(* PLC project HomeAutomation.project, CODESYS CODESYS V3.5 SP21 Patch 3 *)
(* stored: creationDateTime 2026-09-14T20:36:57.2716108, modificationDateTime 2026-09-14T20:35:48.0989634 *)

{attribute 'to_string'}
TYPE E_DIMMER : (idle, soft_turn_on_restore, soft_turn_off, quick_turn_on, quick_turn_off, ramp_up_or_down, low_or_high_entering, low_or_high_leaving, low_or_high_released_by_user, blink);
END_TYPE

TYPE E_DIMMER_CURVE : (linear, logarithmic, cubic);
END_TYPE

(* values of E_RELAY_TYPE: NO: Normally open, and the default. The load is live when the output is TRUE, so a dead PLC leaves it off. What almost every lighting circuit is. Which way round the contact sits decides nothing in the PLC - the output behaves identically either way - and everything in the Home Assistant discovery config, where it swaps the payload_on / payload_off pair so the entity reports the state of the LOAD rather than the state of the coil.; NC: Normally closed. The load is live when the output is FALSE, so a dead PLC leaves it ON - which is the point: sockets, and anything that must survive the controller, are wired this way. Home Assistant reads such an output exactly backwards unless it is told, and no build can catch that, because nothing in the PLC is wrong. *)

{attribute 'qualified_only'}
{attribute 'strict'}
TYPE E_RELAY_TYPE : (NO := 0, NC := 1);
END_TYPE

(* values of E_RS485_DUCO_NODE_TYPE: Unknown: A module type this enumeration does not name, and the value a node holds before the bus has answered for the first time. Zero is deliberately not a Duco type. The manual assigns parameters 01..09 to node 0 and reserves them, so no real component ever reports 0, which leaves it free to mean "not established yet". A node in this state publishes its registers and announces nothing: inventing entities for a component whose layout is unknown would put numbers under labels that were guessed.; DucoBoxFocus: The ventilation unit itself, always node 1. Its register block is the one that is model-specific: read parameters 3, 4 and 5 are current, average and maximum power in watts. A DucoBox Energy or Silent Connect answers those same addresses with something else, which is why this block is named for the Focus.; ValveSensorless: Control valve with no sensor of its own. Reports status, ventilation position and indoor temperature; no CO2 and no humidity.; ValveCO2: Control valve with a CO2 sensor. Adds read parameter 4, the measured CO2 in ppm, and write parameter 1, the CO2 setpoint.; ValveHumidity: Control valve with a humidity sensor. Adds read parameter 5, the relative humidity as a percentage times 100, and write parameters 2 and 3, the RH setpoint and whether delta control is enabled.; UserControl: Wall control, with or without a battery. A battery unit reports no indoor temperature. Its write side collides with the valves': parameters 5 and 6 are the values of buttons 2 and 3 here, where a valve has auto minimum and auto maximum. Anything mapping a holding register to an entity has to branch on the type first.; SensorCO2: CO2 sensor, either a room sensor or a box sensor. A box sensor reports no status and no ventilation position, so its entity set is smaller than a room sensor's even though both answer type 15.; SensorHumidity: Humidity sensor, either a room sensor or a box sensor. Same split as SensorCO2: a box sensor has neither status nor ventilation position.; WindowVentilator: Electronically controlled window ventilator. Two of its registers mean something different from every valve: parameter 2 is the ventilator opening rather than an extraction level, 0 shut to 100 open, and parameter 3 is the OUTDOOR temperature. A reader that assumes "3 is the room temperature" reports the weather as a room.; SwitchSensor: Switch sensor: presence detection, a heat-pump demand input, or an overrule input, selected by write parameter 1. Reports status and ventilation position only.; ActuatorBoard: Actuator board driving a 2/3-point or PWM output. Shares the window ventilator's outdoor temperature on parameter 3, and is the one component where parameter 4 is not CO2 at all: it is the PWM-in percentage. Publishing it as air quality is the mistake this enumeration exists to prevent.; ValveHumidityCO2: Control valve carrying both sensors, and the only type that fills every read parameter: status, position, temperature, CO2 and humidity. Out of sequence at 24 because Duco added it after the 11..19 block was allocated. *)

{attribute 'qualified_only'}
TYPE E_RS485_DUCO_NODE_TYPE : (Unknown := 0, DucoBoxFocus := 10, ValveSensorless := 11, ValveCO2 := 12, ValveHumidity := 13, UserControl := 14, SensorCO2 := 15, SensorHumidity := 16, WindowVentilator := 17, SwitchSensor := 18, ActuatorBoard := 19, ValveHumidityCO2 := 24);
END_TYPE

{attribute 'qualified_only'}
{attribute 'strict'}
{attribute 'to_string'}
TYPE E_HVAC_MODE : (off := 0, auto := 1, heat := 2);
END_TYPE

(* values of E_MQTT_ENTITY: Default: announce as whatever this function block announces by default; Fan: Home Assistant fan platform. Supported by the binary and bistable outputs as an on/off fan; speed and oscillation need topics a binary output has nothing to report on, so they are left out of the published config. *)

{attribute 'qualified_only'}
{attribute 'strict'}
TYPE E_MQTT_ENTITY : (Default := 0, BinarySensor := 1, Sensor := 2, Switch := 3, Light := 4, LightDimmer := 5, Lock := 6, Siren := 7, Valve := 8, Cover := 9, Climate := 10, Event := 11, Fan := 12);
END_TYPE

TYPE MQTT_DISCOVERY_AVTY_T : STRUCT
  topic : JSONVAR;
END_STRUCT;
END_TYPE

TYPE MQTT_DISCOVERY_BASE : STRUCT
  name : JSONVAR;
  default_entity_id : JSONVAR;  (* default entity id *)
  uniq_id : JSONVAR;  (* unique_id *)
  avty : ARRAY[1..2] OF MQTT_DISCOVERY_AVTY_T;  (* availability *)
  avty_mode : JSONVAR;  (* availability mode *)
  pl_avail : JSONVAR;  (* payload_available *)
  pl_not_avail : JSONVAR;  (* payload_not_available *)
  dev : MQTT_DISCOVERY_DEVICE;  (* device *)
  qos : JSONVAR;  (* mqtt qos *)
END_STRUCT;
END_TYPE

TYPE MQTT_DISCOVERY_BINARY_SENSOR : STRUCT
  stat_t : JSONVAR;  (* state_topic *)
  pl_on : JSONVAR;  (* payload_on *)
  pl_off : JSONVAR;  (* payload_off *)
  dev_cla : JSONVAR;  (* device class *)
END_STRUCT;
END_TYPE

TYPE MQTT_DISCOVERY_BINARY_SENSOR_ENT_CAT : STRUCT
  ent_cat : JSONVAR;  (* entity category *)
END_STRUCT;
END_TYPE

TYPE MQTT_DISCOVERY_CLIMATE : STRUCT
  init : JSONVAR;  (* initial desired temperature *)
  curr_temp_t : JSONVAR;  (* current temperature topic *)
  curr_hum_t : JSONVAR;  (* current humidity topic *)
  modes : ARRAY[1..3] OF JSONVAR;  (* modes *)
  mode_cmd_t : JSONVAR;  (* mode command topic *)
  mode_stat_t : JSONVAR;  (* mode state topic *)
  temp_cmd_t : JSONVAR;  (* temperature command topic *)
  temp_stat_t : JSONVAR;  (* temperature state topic *)
  temp_step : JSONVAR;  (* temperature step *)
  opt : JSONVAR;  (* optimistic *)
END_STRUCT;
END_TYPE

TYPE MQTT_DISCOVERY_COVER : STRUCT
  cmd_t : JSONVAR;  (* command_topic *)
  pl_open : JSONVAR;  (* payload open *)
  pl_cls : JSONVAR;  (* payload_close *)
  pl_stop : JSONVAR;  (* payload_stop *)
  stat_t : JSONVAR;  (* state topic *)
  stat_open : JSONVAR;  (* state open *)
  stat_opening : JSONVAR;  (* state opening *)
  stat_clsd : JSONVAR;  (* state closed *)
  stat_closing : JSONVAR;  (* state closing *)
  stat_stopped : JSONVAR;  (* state stopped *)
  opt : JSONVAR;  (* optimistic *)
  dev_cla : JSONVAR;  (* device class *)
END_STRUCT;
END_TYPE

TYPE MQTT_DISCOVERY_COVER_POSITION : STRUCT
  pos_t : JSONVAR;  (* position_topic - where the cover reports how far open it is, as a number between pos_clsd and pos_open. *)
  set_pos_t : JSONVAR;  (* set_position_topic - where Home Assistant asks for a position. Its presence is what puts a slider on the entity rather than three buttons. *)
  pos_open : JSONVAR;  (* position_open - the number that means fully open, normally 100 *)
  pos_clsd : JSONVAR;  (* position_closed - the number that means fully closed, normally 0 *)
END_STRUCT;
END_TYPE

TYPE MQTT_DISCOVERY_DEVICE : STRUCT
  name : JSONVAR;
  cu : JSONVAR;  (* configuration_url *)
  ids : JSONVAR;  (* identifiers *)
  mf : JSONVAR;  (* manufacturer *)
  mdl : JSONVAR;  (* model *)
  sw : JSONVAR;  (* sw_version *)
  hw : JSONVAR;  (* hw_version *)
END_STRUCT;
END_TYPE

TYPE MQTT_DISCOVERY_EVENT : STRUCT
  stat_t : JSONVAR;  (* state topic *)
  evt_typ : ARRAY[1..3] OF JSONVAR;  (* event types *)
  dev_cla : JSONVAR;  (* device class *)
END_STRUCT;
END_TYPE

TYPE MQTT_DISCOVERY_FAN : STRUCT
  cmd_t : JSONVAR;  (* command_topic (REQUIRED) *)
  stat_t : JSONVAR;  (* state_topic *)
  pl_on : JSONVAR;  (* payload_on *)
  pl_off : JSONVAR;  (* payload_off *)
  pct_cmd_t : JSONVAR;  (* percentage_command_topic *)
  pct_stat_t : JSONVAR;  (* percentage_state_topic *)
  spd_rng_min : JSONVAR;  (* speed_range_min *)
  spd_rng_max : JSONVAR;  (* speed_range_max *)
  osc_cmd_t : JSONVAR;  (* oscillation_command_topic *)
  osc_stat_t : JSONVAR;  (* oscillation_state_topic *)
  pl_osc_on : JSONVAR;  (* payload_oscillation_on *)
  pl_osc_off : JSONVAR;  (* payload_oscillation_off *)
  opt : JSONVAR;  (* optimistic *)
END_STRUCT;
END_TYPE

TYPE MQTT_DISCOVERY_LIGHT : STRUCT
  cmd_t : JSONVAR;  (* command_topic *)
  pl_on : JSONVAR;  (* payload_on *)
  pl_off : JSONVAR;  (* payload_off *)
  stat_t : JSONVAR;  (* state_topic *)
  opt : JSONVAR;  (* optimistic *)
END_STRUCT;
END_TYPE

TYPE MQTT_DISCOVERY_LIGHT_DIMMER : STRUCT
  bri_stat_t : JSONVAR;  (* brightness state topic *)
  bri_cmd_t : JSONVAR;  (* brightness command topic *)
  bri_scl : JSONVAR;  (* brightness scale *)
  on_cmd_type : JSONVAR;  (* on command type *)
  dmxChannel : JSONVAR;  (* DMX *)
  dmxWidth : JSONVAR;
  dmxUniverse : JSONVAR;
END_STRUCT;
END_TYPE

TYPE MQTT_DISCOVERY_LOCK : STRUCT
  cmd_t : JSONVAR;  (* command_topic *)
  pl_lock : JSONVAR;  (* payload lock *)
  pl_unlk : JSONVAR;  (* payload unlock *)
  stat_t : JSONVAR;  (* state_topic *)
  stat_locked : JSONVAR;  (* state locked *)
  stat_unlocked : JSONVAR;  (* state unlocked *)
  opt : JSONVAR;  (* optimistic *)
END_STRUCT;
END_TYPE

TYPE MQTT_DISCOVERY_SENSOR : STRUCT
  stat_t : JSONVAR;  (* state_topic *)
  exp_aft : JSONVAR;  (* expire after *)
  dev_cla : JSONVAR;  (* device class, can be null *)
  unit_of_meas : JSONVAR;  (* unit of measurement, can be null *)
  stat_cla : JSONVAR;  (* state class, can be null *)
END_STRUCT;
END_TYPE

TYPE MQTT_DISCOVERY_SENSOR_DIAGNOSTIC : STRUCT
  stat_t : JSONVAR;  (* state_topic *)
  exp_aft : JSONVAR;  (* expire after *)
  ent_cat : JSONVAR;  (* entity category *)
  unit_of_meas : JSONVAR;  (* Added so a diagnostic entity can still carry a unit and keep long-term statistics. A diagnostic sensor is still a sensor: link quality belongs under diagnostics rather than on a dashboard, but it is only worth having if Home Assistant will graph it. Empty on every entity that does not set them, where they serialise as null - the same way stat_cla was added to the ordinary sensor struct. *)
  stat_cla : JSONVAR;
END_STRUCT;
END_TYPE

TYPE MQTT_DISCOVERY_SIREN : STRUCT
  cmd_t : JSONVAR;  (* command_topic *)
  pl_on : JSONVAR;  (* payload_on *)
  pl_off : JSONVAR;  (* payload_off *)
  stat_t : JSONVAR;  (* state_topic *)
  stat_on : JSONVAR;  (* state on *)
  stat_off : JSONVAR;  (* state off *)
  opt : JSONVAR;  (* optimistic *)
END_STRUCT;
END_TYPE

TYPE MQTT_DISCOVERY_SWITCH : STRUCT
  cmd_t : JSONVAR;  (* command_topic *)
  pl_on : JSONVAR;  (* payload_on *)
  pl_off : JSONVAR;  (* payload_off *)
  stat_t : JSONVAR;  (* state_topic *)
  stat_on : JSONVAR;  (* state on *)
  stat_off : JSONVAR;  (* state off *)
  opt : JSONVAR;  (* optimistic *)
  dev_cla : JSONVAR;  (* device class *)
END_STRUCT;
END_TYPE

TYPE MQTT_DISCOVERY_VALVE : STRUCT
  cmd_t : JSONVAR;  (* command topic *)
  pl_open : JSONVAR;  (* payload open *)
  pl_cls : JSONVAR;  (* payload_close *)
END_STRUCT;
END_TYPE

TYPE MQTT_DISCOVERY_VALVE_STATE : STRUCT
  stat_t : JSONVAR;  (* state_topic *)
  stat_clsd : JSONVAR;  (* state clsoed *)
  stat_open : JSONVAR;  (* state closing stat_closing: JSONVAR; state open *)
  opt : JSONVAR;  (* state opening stat_opening: JSONVAR; optimistic *)
  dev_cla : JSONVAR;  (* device class *)
END_STRUCT;
END_TYPE

TYPE ST_MQTT_MESSAGE : STRUCT
  Payload : STRING(1500);
  Topic : STRING(GVL_MQTT.MQTT_TOPIC_LEN);
  Qos : MQTT.QoS;
  MqttRetain : BOOL;
END_STRUCT;
END_TYPE

TYPE MQTT_DISCOVERY_BUTTON : STRUCT
  cmd_t : JSONVAR;  (* command_topic *)
  pl_prs : JSONVAR;  (* payload_press - what is sent when the button is pressed *)
  ent_cat : JSONVAR;  (* entity_category, can be null *)
  dev_cla : JSONVAR;  (* device_class - only identify, restart and update exist for a button; usually null *)
END_STRUCT;
END_TYPE

TYPE MQTT_DISCOVERY_NUMBER : STRUCT
  cmd_t : JSONVAR;  (* command_topic *)
  stat_t : JSONVAR;  (* state_topic - the value the device actually holds, read back rather than assumed *)
  min_val : JSONVAR;  (* min - signed, because a release-the-override value of -1 is a real setting *)
  max_val : JSONVAR;  (* max *)
  step : JSONVAR;  (* step *)
  unit_of_meas : JSONVAR;  (* unit_of_measurement, can be null *)
  mode : JSONVAR;  (* mode - 'box' or 'slider'. A slider on a 0-2000 ppm setpoint is unusable, so this is per entity *)
  dev_cla : JSONVAR;  (* device_class, can be null *)
  ent_cat : JSONVAR;  (* entity_category - 'config' keeps a setpoint out of the main dashboard *)
  opt : JSONVAR;  (* optimistic - FALSE wherever a state topic exists *)
END_STRUCT;
END_TYPE

TYPE A_RS485_READ_BUFFER : ARRAY[0..124] OF WORD;
END_TYPE

TYPE A_RS485_STEP_LIST : ARRAY[0..7] OF ST_RS485_STEP;
END_TYPE

TYPE E_RS485_EASTRON_SDM_DEVICE : (SDM120, SDM220, SDM630);
END_TYPE

(* values of E_RS485_STEP_STATE: IDLE: No step in flight. Start() will be accepted.; BUSY: Transmitting, or waiting for the line to go quiet.; OK: A reply arrived, addressed to us, with the function code we asked for and a CRC of zero over the whole trimmed frame. For a read, ReadBuffer holds Registers() words. Reported for one cycle, then the transport returns to IDLE.; FAILED: No reply, a bad CRC, the wrong slave, the wrong function code, or a Modbus exception reply. Which of those it was is in the transport's counters, not in this value - the scheduler does not need to care and the counters are how a line fault is diagnosed without a scope. *)

{attribute 'qualified_only'}
{attribute 'strict'}
TYPE E_RS485_STEP_STATE : (IDLE := 0, BUSY := 1, OK := 2, FAILED := 3);
END_TYPE

(* values of E_RS485_WORK_LEVEL: NONE: Nothing to do. The scheduler passes over this device.; POLL: A routine read whose interval timer has elapsed. Served round-robin, after every pending COMMAND.; COMMAND: Something a person or Home Assistant asked for, so latency is visible. Served before any POLL, but still round-robin among themselves, so a chatty device cannot starve a quiet one. *)

{attribute 'qualified_only'}
{attribute 'strict'}
TYPE E_RS485_WORK_LEVEL : (NONE := 0, POLL := 1, COMMAND := 2);
END_TYPE

TYPE ST_RS485_COMMISSION_REQUEST : STRUCT
  DeviceId : BYTE;  (* Address the device answers on. Its own, not a guess: a device that has to be hunted for is found by rate and framing, never by walking addresses. *)
  ProbeFunction : BYTE;  (* Function code for the probe read. 3 for holding registers, 4 for input. *)
  ProbeAddress : UINT;  (* Register to read as the probe. Any register that always answers will do - the reply is never decoded, it only has to arrive. *)
  ProbeQuantity : UINT;  (* How many registers the probe asks for. *)
  WriteFunction : BYTE;  (* Function code for the correction. 6 for a single holding register. *)
  WriteAddress : UINT;  (* Register holding the setting that has to change - the device's baud rate, in the only case that exists so far. *)
  WriteValue : WORD;  (* Value that puts the device on this bus. The device encodes it, because only the device knows whether its register takes a rate, a code or an index. *)
  Bauds : ARRAY[0..15] OF UDINT;  (* Rates to try, in the order worth trying them, and how many of them are filled. Put the bus rate first: a device that is already commissioned then costs one Modbus exchange and the sweep ends there. *)
  BaudCount : INT;
  StopBits : ARRAY[0..3] OF BYTE;  (* Framing codes to try, same idea. 255 means leave the port's own framing, which is the ordinary case; 1..3 force the raw SysCom code, because the enumerator names are not portable across runtimes. *)
  StopCount : INT;
  ReportTopic : STRING(32);  (* Topic suffix for the retained result, under the bus prefix. Empty publishes nothing. *)
END_STRUCT;
END_TYPE

TYPE ST_RS485_STEP : STRUCT
  DeviceId : BYTE;  (* Modbus unit id of the slave this step addresses. *)
  FunctionCode : BYTE;  (* 3 read holding, 4 read input, 6 write single, 16 write multiple. Anything else is rejected by the transport rather than guessed at. *)
  Address : UINT;  (* First register, read or write. One field, because a step is only ever one or the other. *)
  Quantity : UINT;  (* Registers to read, or to write. Ignored by FC6, which is always one. *)
  Data : ARRAY[0..7] OF WORD;  (* Payload for a write step. Eight registers is the most an FC16 frame may carry here, which bounds the transmit buffer at 9 + 2*8 = 25 bytes. *)
  AbortOnError : BOOL;  (* TRUE skips the remaining steps of the transaction if this one fails. Set it on the write of a read-after-write: publishing a read-back that never happened, after a write that failed, is the exact inaccuracy the pairing exists to remove. FALSE - the default - suits a batch of independent reads, where one failing register block should not cost the others. *)
END_STRUCT;
END_TYPE

INTERFACE I_RS485_DEVICE
METHOD OnTransactionDone
  VAR_INPUT
    StepsRun : INT;  (* Steps actually executed. Fewer than requested means an AbortOnError step failed. *)
    Failures : INT;  (* How many of those failed. Zero is the only wholly good outcome. *)
  END_VAR
END_METHOD
METHOD OnStepResult
  VAR_INPUT
    StepIndex : INT;  (* Which step of the transaction this is the answer to, indexed as BuildTransaction filled it. Passed in rather than remembered, which is what retires the ActiveRtuQuery and ActiveNode tags every device block used to keep. *)
    Failed : BOOL;  (* No reply, a bad frame, or a Modbus exception. pData holds nothing meaningful. *)
    pData : POINTER TO A_RS485_READ_BUFFER;  (* Registers returned by a read step, big-endian, index 0 being the first register requested. Meaningless for a write step and after a failure. *)
    Count : INT;  (* How many registers pData actually holds. A device that trusts this rather than the quantity it asked for cannot read past the end of a short reply. *)
  END_VAR
END_METHOD
METHOD BuildTransaction : INT
  VAR_INPUT
    pSteps : POINTER TO A_RS485_STEP_LIST;  (* Scheduler-owned scratch. Fill entries 0..n-1 and return n; the memory is only valid for the duration of this call. *)
  END_VAR
END_METHOD
METHOD HasWork : E_RS485_WORK_LEVEL
END_METHOD
METHOD GetCommissioning : BOOL
  VAR_INPUT
    BusBaudrate : UDINT;
    pRequest : POINTER TO ST_RS485_COMMISSION_REQUEST;
  END_VAR
END_METHOD
END_INTERFACE

INTERFACE I_RS485_TRANSPORT
METHOD Registers : INT
END_METHOD
METHOD ReadBuffer : POINTER TO A_RS485_READ_BUFFER
END_METHOD
METHOD Service : E_RS485_STEP_STATE
END_METHOD
METHOD Start : BOOL
  VAR_INPUT
    pStep : POINTER TO ST_RS485_STEP;
  END_VAR
END_METHOD
METHOD Retune : BOOL
  VAR_INPUT
    Baudrate : UDINT;  (* 0 keeps the configured rate *)
    StopBitsRaw : BYTE;  (* 255 keeps the configured framing *)
    ReplyTimeout : TIME;  (* T#0S keeps the configured timeout *)
    GapTime : TIME;  (* T#0S keeps the configured gap *)
  END_VAR
END_METHOD
METHOD RestoreTuning
END_METHOD
METHOD LastRxCount : UDINT
END_METHOD
END_INTERFACE

{attribute 'reflection'}
FUNCTION_BLOCK FB_INPUT_BINARYSENSOR_MQTT EXTENDS FB_MQTT_BASE
  VAR_OUTPUT
    Q : BOOL;  (* Follows the input but debounced *)
    EVENT : BOOL;  (* Event outputs only high for on clock cycle *)
    EVENT_R : BOOL;
    EVENT_F : BOOL;
  END_VAR
  VAR
    {attribute 'noinit'}
    {attribute 'instance-path'}
    sInstancePath : STRING(GVL_MQTT.MQTT_TOPIC_LEN);  (* object's full instance name *)
    bStartup : BOOL := TRUE;
    fbDebounce : OSCAT_BUILDING.DEBOUNCE;  (* to debounce the physical input *)
    fbRTrig : Standard.R_TRIG;  (* to detect a rising edge on the debounced signal *)
    fbFTrig : Standard.F_TRIG;  (* to detect a falling edge on the debounced signal *)
    T_TurnOffDelay : TIME := TIME#0ms;
    fbTurnOffDelayTimer : OSCAT_BASIC.TOF;
  END_VAR
  VAR_INPUT
    BS : BOOL;
    ProcessImageValid : BOOL := TRUE;  (* TRUE once the K-bus has finished starting and the mapped inputs mean something. FALSE holds this sensor at rest. Defaulted TRUE so no existing call site changes behaviour, but pass Pfc200Bus.xConfigFinished on anything whose loop is normally CLOSED. Until the bus is up every mapped word reads zero, and on an inverted loop zero IS the alarm - so a fire sensor left ungated raises its alarm on every single cold start, deterministically. That is not a plausible-looking value like an RTD's 0.0 C; it is the tripped state itself. *)
  END_VAR

            (* --- self-wiring prologue ----------------------------------------------------
   Makes the InitMqtt and InitMqttDiscovery* calls optional. Set FriendlyName at
   the declaration site and this block wires itself from GVL_MQTT on its
   first cyclic call, then announces itself to Home Assistant.

   Deliberately in the body rather than in FB_init: it dereferences GVL members
   and reads the reflection instance path, and doing that during initialisation
   would rely on an ordering nothing enforces and the compiler cannot check. The
   body is the same lifecycle phase the init actions used, so this is not merely
   safe, it is the phase that already works today.

   The wiring calls this block's own unmodified InitMqtt / InitMqttDiscovery*
   methods, so anything published - topics and discovery JSON alike - is produced
   by exactly the code that produces it today. Only the trigger moved.

   Dormant while FriendlyName is empty, so existing projects and existing call
   sites keep working untouched.

   A block wired this way MUST be called cyclically. An instance whose body never
   runs is now unwired and absent from Home Assistant, where the init action used
   to wire it regardless. Nothing warns about that.  *)
IF FriendlyName <> '' THEN

	IF NOT bInitMqttDone THEN
		THIS^.InitMqtt(
			MQTTPublishPrefix := ADR(GVL_MQTT.MqttPushbuttonPrefix),
			pMqttPublishQueue := ADR(GVL_MQTT.fbMqttPublishQueue));
	END_IF

	IF bInitMqttDone AND NOT bInitMqttDiscoveryDone THEN
		THIS^.InitMqttDiscovery(
			Device := ADR(GVL_MQTT.PLC_Device),
			Name := FriendlyName);
	END_IF

END_IF

(* Held at rest until the process image is valid. The debounce below then
   still has to settle, so a genuine alarm present at power-up is reported a
   few cycles late rather than not at all. *)
fbDebounce(IN := BS AND ProcessImageValid,	
	TD := T#50MS, (* 2x cyle + 10ms *)
	PM := FALSE
	);
	
fbTurnOffDelayTimer(IN:=fbDebounce.Q,
	PT := T_TurnOffDelay,
	Q=>Q
	);

fbRTrig(CLK := fbTurnOffDelayTimer.Q);
fbFTrig(CLK := fbTurnOffDelayTimer.Q);

EVENT := fbRTrig.Q OR fbFTrig.Q;
EVENT_R := fbRTrig.Q;
EVENT_F := fbFTrig.Q;

IF (fbRTrig.Q OR (bStartup AND fbDebounce.Q)) AND bInitMqttDone THEN
	pMqttPublishQueue^.AddMessage(
		Payload := 'ON',
		Topic := CONCAT(psMqttPublishTopicPrefix^, MqttPublishTopicSuffix),
		Qos := MQTT.QoS.ExactlyOnce,
		MqttRetain := TRUE
	);
	bStartup:=FALSE;	
END_IF

IF (fbFTrig.Q OR (bStartup AND NOT(fbDebounce.Q))) AND bInitMqttDone THEN
	pMqttPublishQueue^.AddMessage(
		Payload := 'OFF',
		Topic := CONCAT(psMqttPublishTopicPrefix^, MqttPublishTopicSuffix),
		Qos := MQTT.QoS.ExactlyOnce,
		MqttRetain := TRUE
	);
	bStartup:=FALSE;	
END_IF
          

METHOD ConfigureFunctionBlock
  VAR_INPUT
    T_TurnOffDelay : TIME;
  END_VAR
                  THIS^.T_TurnOffDelay:=T_TurnOffDelay;
                
END_METHOD

METHOD InitMqttDiscovery
  VAR_INPUT
    Device : POINTER TO FB_PLC_MQTT_DISCOVERY_DEVICE;
    Name : STRING(255);
    DeviceClass : STRING(100) := 'smoke';
    overruleId : STRING(255) := '';
  END_VAR
  VAR
    id : STRING(255);
  END_VAR
                  IF bInitMqttDone AND NOT bInitMqttDiscoveryDone THEN
	
	id := SUPER^.ResolveEntityId(overruleId);
	
	Device^.CreateBinarySensorEntity(
		Id := id,
		Name := name,
		StateTopic := THIS^.sMQTTPublishTopic,
		PayloadOn := 'ON',
		PayloadOff := 'OFF',
		DeviceClass := DeviceClass);
		
	bInitMqttDiscoveryDone := TRUE;
END_IF		
                
END_METHOD

METHOD InitMqtt
  VAR_INPUT
    MQTTPublishPrefix : POINTER TO STRING;
    pMqttPublishQueue : POINTER TO FB_MQTT_PUBLISH_QUEUE;
  END_VAR
                  SUPER^._sInstancePath := THIS^.sInstancePath; // Due to reflection its location is important

(*pass trough*)
THIS^.pMqttPublishQueue := pMqttPublishQueue;
THIS^.psMqttPublishTopicPrefix:=MQTTPublishPrefix;
SUPER^.InitBaseMqtt();

                
END_METHOD
END_FUNCTION_BLOCK

{attribute 'reflection'}
FUNCTION_BLOCK FB_INPUT_PUSHBUTTON_DIMMER_MQTT EXTENDS FB_MQTT_BASE
  VAR_OUTPUT
    DIM : BYTE;
    DBL : BOOL;
    Q : BOOL;
    SINGLE : BOOL;
    DOUBLE : BOOL;
    LONG : BOOL;
    P_LONG : BOOL;
  END_VAR
  VAR
    {attribute 'noinit'}
    {attribute 'instance-path'}
    sInstancePath : STRING(GVL_MQTT.MQTT_TOPIC_LEN);  (* object's full instance name *)
    fbDimmer : OSCAT_BUILDING.DIMM_I;
    OutputDimmer : BOOL;
    Qos_Dimm : MQTT.QoS;
    Delta_Dimm : INT;
    fbDetectpush : OSCAT_BUILDING.CLICK_MODE;
    fbPLongRTrig : Standard.R_TRIG;
    fbPLongFTrig : Standard.F_TRIG;
    byPreviousDim : BYTE;  (* Vars to detect statechanges on outputs *)
    bPreviousQ : BOOL;
    bPreviousDBL : BOOL;
    T_Debounce : TIME := TIME#10ms;  (* Default values for E_DIMMER, can be overwritten by method call *)
    T_Reconfig : TIME := TIME#10s0ms;
    T_On_Max : TIME := TIME#0ms;
    T_Dimm_Start : TIME := TIME#400ms;
    T_Dimm : TIME := TIME#3s0ms;
    Min_On : BYTE := 50;
    Max_On : BYTE := 255;
    Soft_Dimm : BOOL := TRUE;
    Dbl_Toggle : BOOL := FALSE;
    Rst_Out : BOOL := FALSE;
    T_Long : TIME := TIME#400ms;  (* Default value for click mode, can be overwritten by method call *)
  END_VAR
  VAR_INPUT
    PB : BOOL;
    SET : BOOL;
    VAL : BYTE;
    RST : BOOL;
  END_VAR
  VAR
    bDimPublished : BOOL;  (* TRUE once the dim level has been published at least once. Without it a freshly discovered sensor sits at "unknown" until somebody touches the pushbutton, because a level that has not moved is never published. *)
  END_VAR

            (* --- self-wiring prologue ----------------------------------------------------
   Makes the InitMqtt and InitMqttDiscovery calls optional. Set FriendlyName at
   the declaration site and this block wires itself from GVL_MQTT on its first
   cyclic call, then announces itself to Home Assistant.

   Deliberately in the body rather than in FB_init: it dereferences GVL members
   and reads the reflection instance path, and doing that during initialisation
   would rely on an ordering nothing enforces and the compiler cannot check.

   Dormant while FriendlyName is empty, so existing call sites that still make
   the explicit InitMqtt call keep working untouched.

   A block wired this way MUST be called cyclically. An instance whose body never
   runs is now unwired and absent from Home Assistant, where an init action used
   to wire it regardless. Nothing warns about that. *)
IF FriendlyName <> '' THEN

	IF NOT bInitMqttDone THEN
		THIS^.InitMqtt(
			MQTTPublishPrefix := ADR(GVL_MQTT.MqttPushbuttonPrefix),
			pMqttPublishQueue := ADR(GVL_MQTT.fbMqttPublishQueue),
			OutputDimmer := TRUE,
			Qos_Dimm := MQTT.QoS.ExactlyOnce,
			Delta_Dimm := 5);
	END_IF

	IF bInitMqttDone AND NOT bInitMqttDiscoveryDone THEN
		THIS^.InitMqttDiscovery(
			Device := ADR(GVL_MQTT.PLC_Device),
			Name := FriendlyName);
	END_IF

END_IF

fbDimmer(
	IN:= PB,
	SET:= SET,
	VAL:= VAL,
	RST:= RST,
	OUT:= DIM,
	T_DEBOUNCE:= T_Debounce,
	T_RECONFIG:= T_Reconfig,
	T_ON_MAX:= T_On_Max,
	T_DIMM_START:= T_Dimm_Start,
	T_DIMM:= T_Dimm,
	MIN_ON:= Min_On,
	MAX_ON:= Max_On,
	SOFT_DIMM:= Soft_Dimm,
	DBL_TOGGLE:= Dbl_Toggle,
	RST_OUT:= Rst_Out,
	Q=> Q,
	DBL=> DBL);
	
fbDetectpush(
	IN:= PB, 	
	SINGLE=> SINGLE, 
	DOUBLE=> DOUBLE, 
	TP_LONG=> LONG, 
	T_LONG:= T_long);
	
fbPLongRTrig(CLK:=fbDetectpush.LONG);
fbPLongFTrig(CLK:=fbDetectpush.LONG);

(* The dim level is state, not an event, so it is published retained: after a
   Home Assistant restart the sensor gets its value back from the broker instead
   of reading "unknown" until somebody dims something.

   Published once as soon as MQTT is up, whatever it reads, so a newly
   discovered entity has a value at all - a level that has not moved would
   otherwise never be published. After that it is Delta_Dimm that decides, with
   the value on release always sent so MQTT and the output cannot drift apart.

   Qos_Dimm is the QoS for this stream, which is what its name and the
   documentation have always said; it used to be applied to Q instead. *)
IF bInitMqttDone AND OutputDimmer
	AND (NOT bDimPublished
		OR ((ABS(BYTE_TO_INT(byPreviousDim) - BYTE_TO_INT(DIM)) >= Delta_Dimm OR PB = FALSE) AND DIM <> byPreviousDim)) THEN
	byPreviousDim := DIM;
	bDimPublished := TRUE;
	pMqttPublishQueue^.AddMessage(		
		Payload := BYTE_TO_STRING(DIM),
		Topic := CONCAT(sMQTTPublishTopic, '/DIM'),
		Qos := Qos_Dimm,
		MqttRetain := TRUE
	);
END_IF

IF fbDimmer.Q <> bPreviousQ AND bInitMqttDone THEN
	bPreviousQ:=fbDimmer.Q;
	pMqttPublishQueue^.AddMessage(
		Payload := BOOL_TO_STRING(fbDimmer.Q),
		Topic := CONCAT(sMQTTPublishTopic, '/Q'),
		Qos := MQTT.QoS.ExactlyOnce,
		MqttRetain := TRUE
	);
END_IF

IF fbDimmer.DBL <> bPreviousDBL AND bInitMqttDone THEN
	bPreviousDBL:=fbDimmer.DBL;
	pMqttPublishQueue^.AddMessage(
		Payload := BOOL_TO_STRING(fbDimmer.DBL),
		Topic := CONCAT(sMQTTPublishTopic, '/DBL'),
		Qos := MQTT.QoS.ExactlyOnce,
		MqttRetain := TRUE
	);
END_IF

(* The three press payloads are JSON because the entity announced for them is a
   Home Assistant event entity, which reads event_type out of the payload. A
   bare 'SINGLE' would arrive and be discarded. *)
IF fbDetectpush.SINGLE AND bInitMqttDone THEN
	pMqttPublishQueue^.AddMessage(
		Payload := '{"event_type": "SINGLE"}',
		Topic := sMQTTPublishTopic,
		Qos := MQTT.QoS.ExactlyOnce,
		MqttRetain := FALSE
	);
END_IF

IF fbDetectpush.DOUBLE AND bInitMqttDone THEN
	pMqttPublishQueue^.AddMessage(
		Payload := '{"event_type": "DOUBLE"}',
		Topic := sMQTTPublishTopic,
		Qos := MQTT.QoS.ExactlyOnce,
		MqttRetain := FALSE
	);
END_IF

IF fbDetectpush.TP_LONG AND bInitMqttDone THEN
	pMqttPublishQueue^.AddMessage(
		Payload := '{"event_type": "LONG"}',
		Topic := sMQTTPublishTopic,
		Qos := MQTT.QoS.ExactlyOnce,
		MqttRetain := FALSE
	);
END_IF

IF (fbPLongRTrig.Q OR fbPLongFTrig.Q) AND bInitMqttDone THEN
	pMqttPublishQueue^.AddMessage(
		Payload := BOOL_TO_STRING(fbDetectpush.LONG),
		Topic := CONCAT(sMQTTPublishTopic,'/P_LONG'),
		Qos := MQTT.QoS.ExactlyOnce,
		MqttRetain := TRUE
	);
END_IF

          

METHOD ConfigureFunctionBlock
  VAR_INPUT
    T_Debounce : TIME;  (* Default values for E_DIMMER, can be overwritten by method call *)
    T_Reconfig : TIME;
    T_On_Max : TIME;
    T_Dimm_Start : TIME;
    T_Dimm : TIME;
    Min_On : BYTE;
    Max_On : BYTE;
    Soft_Dimm : BOOL;
    Dbl_Toggle : BOOL;
    Rst_Out : BOOL;
    T_Long : TIME;  (* Default value for click mode, can be overwritten by method call *)
  END_VAR
                  THIS^.T_Debounce:=T_Debounce;
THIS^.T_Reconfig:=T_Reconfig;
THIS^.T_On_Max:=T_On_Max;
THIS^.T_Dimm_Start:=T_Dimm_Start;
THIS^.T_Dimm:=T_Dimm;
THIS^.Min_On:=Min_On;
THIS^.Max_On:=Max_On;
THIS^.Soft_Dimm:=Soft_Dimm;
THIS^.Dbl_Toggle:=Dbl_Toggle;
THIS^.Rst_Out:=Rst_Out;

THIS^.T_Long:=T_Long;
                
END_METHOD

METHOD InitMqtt
  VAR_INPUT
    MQTTPublishPrefix : POINTER TO STRING;
    pMqttPublishQueue : POINTER TO FB_MQTT_PUBLISH_QUEUE;
    OutputDimmer : BOOL;
    Qos_Dimm : MQTT.QoS;
    Delta_Dimm : INT;
  END_VAR
                  SUPER^._sInstancePath := THIS^.sInstancePath; // Due to reflection its location is important

(*pass trough*)
THIS^.pMqttPublishQueue := pMqttPublishQueue;
THIS^.psMqttPublishTopicPrefix := MQTTPublishPrefix;
SUPER^.InitBaseMqtt();

THIS^.OutputDimmer:=OutputDimmer;
THIS^.Qos_Dimm:=Qos_Dimm;
THIS^.Delta_Dimm:=Delta_Dimm;
                
END_METHOD

METHOD InitMqttDiscovery
  VAR_INPUT
    Device : POINTER TO FB_PLC_MQTT_DISCOVERY_DEVICE;
    Name : STRING(255);
    overruleId : STRING(255) := '';
  END_VAR
  VAR
    id : STRING(255);
    eventTypes : ARRAY[1..3] OF STRING := ['SINGLE', 'DOUBLE', 'LONG'];
  END_VAR
                  (* Two entities, because this block is two things on one topic tree: a wall
   pushbutton and a dim level.

   The button is announced exactly as FB_INPUT_PUSHBUTTON_MQTT announces one -
   an event entity carrying SINGLE, DOUBLE and LONG. That is why the three
   press payloads below are JSON: Home Assistant's event platform reads
   event_type out of the payload, and a bare 'SINGLE' is not a payload it can
   read.

   The level is a sensor, not a light. A light entity would have to be
   commandable, and this block has no subscribe side at all - no callback
   collector, no command topics. FB_OUTPUT_DIMMER_MQTT is the block that does
   have those, and it is what to reach for when Home Assistant has to set the
   level rather than watch it.

   ExpiryAfter is 0 on purpose. There is no heartbeat here: DIM publishes on
   change, gated by Delta_Dimm, so any positive expiry would grey out a level
   that is merely steady.

   No per-entity availability topic either. Nothing in this block can be
   individually untrustworthy the way an RTD channel can, so both availability
   slots stay with the PLC device. *)
IF bInitMqttDone AND NOT bInitMqttDiscoveryDone THEN

	id := SUPER^.ResolveEntityId(overruleId);

	Device^.CreateEventEntity(
		Name := Name,
		Id := id,
		StateTopic := THIS^.sMQTTPublishTopic,
		EventTypes := eventTypes,
		Deviceclass := 'button');

	Device^.CreateSensorEntity(
		Name := CONCAT(Name, ' level'),
		Id := CONCAT(id, '_DIM'),
		StateTopic := CONCAT(THIS^.sMQTTPublishTopic, '/DIM'),
		ExpiryAfter := 0);

	bInitMqttDiscoveryDone := TRUE;
END_IF
                
END_METHOD
END_FUNCTION_BLOCK

{attribute 'reflection'}
FUNCTION_BLOCK FB_INPUT_PUSHBUTTON_MQTT EXTENDS FB_MQTT_BASE
  VAR_OUTPUT
    SINGLE : BOOL;
    DOUBLE : BOOL;
    LONG : BOOL;
    P_LONG : BOOL;
  END_VAR
  VAR
    {attribute 'noinit'}
    {attribute 'instance-path'}
    sInstancePath : STRING(GVL_MQTT.MQTT_TOPIC_LEN);  (* Refelection: object's full instance name *)
    fbDetectpush : OSCAT_BUILDING.CLICK_MODE;
    fbPLongRTrig : Standard.R_TRIG;
    fbPLongFTrig : Standard.F_TRIG;
    T_Long : TIME := TIME#400ms;  (* Default value for click mode, can be overwritten by method call *)
  END_VAR
  VAR_INPUT
    PB : BOOL;
  END_VAR

            (* --- self-wiring prologue ----------------------------------------------------
   Makes the InitMqtt and InitMqttDiscovery* calls optional. Set FriendlyName at
   the declaration site and this block wires itself from GVL_MQTT on its
   first cyclic call, then announces itself to Home Assistant.

   Deliberately in the body rather than in FB_init: it dereferences GVL members
   and reads the reflection instance path, and doing that during initialisation
   would rely on an ordering nothing enforces and the compiler cannot check. The
   body is the same lifecycle phase the init actions used, so this is not merely
   safe, it is the phase that already works today.

   The wiring calls this block's own unmodified InitMqtt / InitMqttDiscovery*
   methods, so anything published - topics and discovery JSON alike - is produced
   by exactly the code that produces it today. Only the trigger moved.

   Dormant while FriendlyName is empty, so existing projects and existing call
   sites keep working untouched.

   A block wired this way MUST be called cyclically. An instance whose body never
   runs is now unwired and absent from Home Assistant, where the init action used
   to wire it regardless. Nothing warns about that.  *)
IF FriendlyName <> '' THEN

	IF NOT bInitMqttDone THEN
		THIS^.InitMqtt(
			MQTTPublishPrefix := ADR(GVL_MQTT.MqttPushbuttonPrefix),
			pMqttPublishQueue := ADR(GVL_MQTT.fbMqttPublishQueue));
	END_IF

	IF bInitMqttDone AND NOT bInitMqttDiscoveryDone THEN
		THIS^.InitMqttDiscovery(
			Device := ADR(GVL_MQTT.PLC_Device),
			Name := FriendlyName);
	END_IF

END_IF

fbDetectpush(
	IN:= PB, 	
	SINGLE=> SINGLE, 
	DOUBLE=> DOUBLE, 
	TP_LONG=> LONG, 
	LONG=> P_LONG,
	T_LONG:= T_Long);
	
fbPLongRTrig(CLK:=fbDetectpush.LONG);
fbPLongFTrig(CLK:=fbDetectpush.LONG);
	
IF fbDetectpush.SINGLE AND bInitMqttDone THEN
	pMqttPublishQueue^.AddMessage(
		Payload := '{"event_type": "SINGLE"}',
		Topic := CONCAT(psMqttPublishTopicPrefix^, MqttPublishTopicSuffix),
		Qos := MQTT.QoS.ExactlyOnce,
		MqttRetain := FALSE
	);
END_IF

IF fbDetectpush.DOUBLE AND bInitMqttDone THEN
	pMqttPublishQueue^.AddMessage(
		Payload := '{"event_type": "DOUBLE"}',
		Topic := CONCAT(psMqttPublishTopicPrefix^, MqttPublishTopicSuffix),
		Qos := MQTT.QoS.ExactlyOnce,
		MqttRetain := FALSE
	);
END_IF

IF fbDetectpush.TP_LONG AND bInitMqttDone THEN
	pMqttPublishQueue^.AddMessage(
		Payload := '{"event_type": "LONG"}',
		Topic := sMQTTPublishTopic,
		Qos := MQTT.QoS.ExactlyOnce,
		MqttRetain := FALSE
	);
END_IF
          

METHOD ConfigureFunctionBlock
  VAR_INPUT
    T_Long : TIME;  (* Default value for click mode, can be overwritten by method call *)
  END_VAR
                  THIS^.T_Long:=T_Long;
                
END_METHOD

METHOD InitMqtt
  VAR_INPUT
    MQTTPublishPrefix : POINTER TO STRING;
    pMqttPublishQueue : POINTER TO FB_MQTT_PUBLISH_QUEUE;
  END_VAR
                  SUPER^._sInstancePath := THIS^.sInstancePath; // Due to reflection its location is important

(*pass trough*)
THIS^.pMqttPublishQueue := pMqttPublishQueue;
THIS^.psMqttPublishTopicPrefix:=MQTTPublishPrefix;
SUPER^.InitBaseMqtt();

                
END_METHOD

METHOD InitMqttDiscovery
  VAR_INPUT
    Device : POINTER TO FB_PLC_MQTT_DISCOVERY_DEVICE;
    Name : STRING(255);
    overruleId : STRING(255) := '';
  END_VAR
  VAR
    id : STRING(255);
    eventTypes : ARRAY[1..3] OF STRING := ['SINGLE', 'DOUBLE', 'LONG'];
  END_VAR
                  IF bInitMqttDone AND NOT bInitMqttDiscoveryDone THEN
	
	id := SUPER^.ResolveEntityId(overruleId);
	
	Device^.CreateEventEntity(
		Name := name,
		Id := id,
		StateTopic := THIS^.sMQTTPublishTopic,
		EventTypes := eventTypes,
		Deviceclass := 'button');

	bInitMqttDiscoveryDone := TRUE;
END_IF		
                
END_METHOD
END_FUNCTION_BLOCK

{attribute 'reflection'}
FUNCTION_BLOCK FB_INPUT_TEMPERATURE_RTD_MQTT EXTENDS FB_MQTT_BASE
  VAR_OUTPUT
    Temperature : REAL;  (* Degrees Celsius. Held at the last trustworthy reading while Fault is set, rather than following the channel into whatever it reports for a broken wire. *)
    Valid : BOOL;  (* The channel is reading a real sensor, within what the sensor type can measure AND within what this sensor could plausibly be measuring. *)
    Fault : BOOL;  (* Do not trust this reading. Set when the value is outside what the sensor type can physically produce, and when the channel has gone StaleTimeout without moving a digit, and when it is outside PlausibleMin..PlausibleMax. This is what drives the entity's availability: while it is set, Home Assistant shows the sensor as unavailable. *)
    DataAvailable : BOOL;  (* High once a plausible reading has been seen, and it latches. It answers "has this channel ever worked", not "is it working now" - Valid is that one. One wart, found by a bench assertion that expected better: a mapped channel reads 0 for the first cycles, before the K-bus has filled the process image, and 0.0 C is a perfectly plausible reading. So this latches TRUE - and Temperature holds 0.0 - even on a channel that goes on to measure nothing at all. Do not read it as proof a sensor is connected. *)
  END_VAR
  VAR
    {attribute 'noinit'}
    {attribute 'instance-path'}
    sInstancePath : STRING;  (* object's full instance name *)
    fbFirstConversion : Standard.TON;
    bZeroIsBelievable : BOOL;  (* FALSE only in the moments after the bus comes up, while the channel still reads the zero the process image was cleared to. *)
    iPublishedRaw : INT;  (* The channel word as it was last published, so a repeat can be told from a change. Kept as the INT rather than the REAL: two readings that came from the same word are then equal by construction, with no float comparison. *)
    bPublishedValid : BOOL;
    fbHeartbeat : Standard.TON;
    fbFaultEdge : Standard.R_TRIG;
    fbHealEdge : Standard.F_TRIG;
    bStartup : BOOL := TRUE;
    bInRange : BOOL;
    bPlausible : BOOL;
    rReading : REAL;
    sPayload : STRING(20);
    iWhole : INT;
    iTenth : INT;
    iLeadOffset : INT;  (* LeadResistance expressed in the module's own units - tenths of a degree. *)
    iCorrectedRaw : INT;  (* Raw with the lead correction taken off. Everything downstream reads this rather than Raw, except the movement check. *)
  END_VAR
  VAR CONSTANT
    ciRtdMinRaw : INT := -2000;  (* What a platinum RTD can physically report, per IEC 60751: -200 C to 850 C. Anything outside it is the module telling you about the wiring rather than the temperature, whatever value it happens to use to say so - which is why the check is a range in engineering units and not a magic fault code. *)
    ciRtdMaxRaw : INT := 8500;
    ctFirstConversion : TIME := TIME#5s0ms;  (* How long a channel may read exactly 0 after the bus comes up before 0 is believed as a temperature. ProcessImageValid is necessary and NOT sufficient: the bus reports process data exchanging a little before an RTD module has delivered its first conversion, and in that window the word is still the zeroed process image. Measured on the bench, that window is well under a second - but 0 is 0.0 C, a perfectly plausible temperature, so a block that believes it publishes a fabricated zero on every restart. Long enough for any 750-series RTD to convert, short enough that a sensor genuinely sitting at 0.0 C is only briefly unavailable rather than wrong. *)
    crPt1000OhmsPerDegree : REAL := 3.9;  (* dR/dT of a Pt1000 near room temperature, per IEC 60751. The local slope at 0 C is 3.9083; 3.85 is the mean coefficient over 0..100 C and is the wrong number here, because a lead correction is applied where the sensor is, not averaged over its whole span. *)
  END_VAR
  VAR_INPUT
    Raw : INT;  (* The mapped channel word of an RTD input module, in tenths of a degree Celsius - which is what a WAGO 750-463 and its relatives put in the process image, two's complement, so -105 is -10.5 C. Wire it straight to the channel variable: Raw := RTD_001. *)
    ProcessImageValid : BOOL := FALSE;  (* TRUE once the K-bus has finished starting and is really exchanging process data. Until then every mapped word reads 0, and 0 is 0.0 C - a perfectly plausible temperature - so a block that trusts it publishes a fabricated zero on every restart before the real value arrives a second later. That happened, on this bench, and it is why this input exists. Wire it to the bus driver's own answer, which is the only authoritative one: ProcessImageValid := Pfc200Bus.xConfigFinished. Defaults to FALSE, deliberately. Forget to wire it and the channel stays unavailable, which is loud; the alternative default hands you a wrong number once per restart, which is silent. *)
    LeadResistance : REAL := 0.0;  (* Round-trip resistance of the sensor leads, in ohms. Zero, and nothing is corrected. A 750-451 and a 750-463 both measure 2-conductor, so nothing compensates for the wire: the leads sit in series with the element and the channel reads HIGH by them. Near room temperature a Pt1000 moves about 3.9 ohms per degree, so the error is LeadResistance / 3.9 degrees - about 0.18 C down 2x10 m of 0.5 mm2, and 1.8 C down 2x50 m of 0.25 mm2. Ignorable on a bench, not ignorable on a long run. Measure it with the sensor disconnected, by shorting the far end of the pair and reading the loop at the terminals. CORRECT THIS IN ONE PLACE ONLY. The module carries its own user scaling and user calibration, written with WAGO-I/O-CHECK and unreadable from CODESYS - set an offset there as well and it is applied twice, with nothing anywhere to say so. Prefer here: this is in source control, it shows up in a diff and in the PLCopen export, and it survives swapping the terminal, which a value in a module's flash does not. *)
    HeartbeatInterval : TIME := TIME#1m0s0ms;  (* Republish even when nothing changed, so a reader can tell a steady temperature from a PLC that has stopped. Paired with the discovery config's expire_after, which is set to three of these - so a minute here means Home Assistant gives up on a silent channel after three. *)
    PlausibleMin : REAL := -40.0;  (* The range this sensor could plausibly be measuring, in degrees Celsius. The IEC 60751 bounds only ask whether a platinum RTD could produce a reading at all, which turns out to be a very weak question: a WAGO 750-463 reports an open circuit as 150.0 C, a legal Pt1000 temperature that passes the range check and publishes as healthy until StaleTimeout eventually notices. No room, buffer tank or floor loop reaches 150 C, so saying what this sensor is for rejects that on the first scan instead of a quarter of an hour later. Widen it deliberately for a flue, a solar collector or a freezer. Set Max <= Min to switch the check off. *)
    PlausibleMax : REAL := 80.0;
  END_VAR

            (* --- self-wiring prologue ----------------------------------------------------
   Set FriendlyName at the declaration and this block wires itself from GVL_MQTT
   on its first cyclic call, then announces itself to Home Assistant. Same idiom,
   and the same reasons, as every other block here: see
   FB_INPUT_BINARYSENSOR_MQTT.

   A block wired this way MUST be called cyclically. An instance whose body never
   runs stays unwired and never appears in Home Assistant, and nothing warns
   about it. *)
IF FriendlyName <> '' THEN

	IF NOT bInitMqttDone THEN
		THIS^.InitMqtt(
			MQTTPublishPrefix := ADR(GVL_MQTT.MqttPubAnalogInputPrefix),
			pMqttPublishQueue := ADR(GVL_MQTT.fbMqttPublishQueue));
	END_IF

	IF bInitMqttDone AND NOT bInitMqttDiscoveryDone THEN
		THIS^.InitMqttDiscovery(
			Device := ADR(GVL_MQTT.PLC_Device),
			Name := FriendlyName);
	END_IF

END_IF

(* --- is this a temperature, and is it a temperature THIS sensor could see? ---
   Two bounds, answering two different questions, and only the second one is
   much use on real hardware.

   ciRtdMinRaw/MaxRaw is IEC 60751: what a platinum RTD can physically report at
   all. Anything outside it is the module talking about the wiring rather than
   the temperature, whatever value it picks to say so.

   PlausibleMin/Max is what this particular sensor could be measuring, and it is
   the check that catches the failure this block actually met. A WAGO 750-463
   reports an open circuit as 150.0 C - a perfectly legal Pt1000 temperature,
   inside IEC 60751, which sailed through the range check and published as a
   healthy reading for the fifteen minutes it took StaleTimeout to notice. No
   room, buffer tank or floor loop ever reaches 150 C. Saying so rejects it on
   the first scan. *)
(* --- lead resistance, on a module that cannot compensate for it --------------
   2-conductor measurement puts the leads in series with the element, so the
   channel reads high by LeadResistance / 3.9 degrees. Corrected here, in tenths
   and in integers, so the single decimal the module actually has reaches the
   payload unchanged rather than through a REAL round trip.

   Zero by default and REAL_TO_INT(0.0) is 0, so a channel that names no lead
   resistance behaves exactly as it did before this existed. *)
iLeadOffset := REAL_TO_INT(LeadResistance / crPt1000OhmsPerDegree * 10.0);
iCorrectedRaw := Raw - iLeadOffset;

bInRange := (iCorrectedRaw >= ciRtdMinRaw) AND (iCorrectedRaw <= ciRtdMaxRaw);
(* Tenths of a degree, so the scaling is exact rather than a calibration. *)
rReading := INT_TO_REAL(iCorrectedRaw) / 10.0;
bPlausible := (PlausibleMax <= PlausibleMin)
	OR ((rReading >= PlausibleMin) AND (rReading <= PlausibleMax));
(* --- has this channel produced a reading at all? -----------------------------
   Two gates before the value is looked at, because a zero has two meanings.

   ProcessImageValid says the bus is exchanging process data. Necessary, and NOT
   sufficient: it goes TRUE slightly before an RTD module has delivered its first
   conversion, and until then the word is still the zero the process image was
   cleared to. That gap is well under a second and it was enough to publish a
   fabricated 0.0 C on every restart, ahead of the real value.

   So a zero is not believed until the module has had time to convert. After
   ctFirstConversion it is believed like any other reading, because 0.0 C is a
   real temperature and a sensor sitting at it must not go unavailable forever.
   Raw and not iCorrectedRaw: it is the module's own word that is zeroed, and a
   lead correction would move it off zero for the wrong reason. *)
fbFirstConversion(IN := ProcessImageValid, PT := ctFirstConversion);
bZeroIsBelievable := (Raw <> 0) OR fbFirstConversion.Q;

Valid := ProcessImageValid AND bZeroIsBelievable AND bInRange AND bPlausible;

IF Valid THEN
	Temperature := rReading;
	DataAvailable := TRUE;
END_IF

(* Out of range or implausible is the whole of the fault surface. There was a
   movement check here too - a channel that had not changed a digit for
   StaleTimeout was called Stuck and faulted - and it was removed because it does
   not survive contact with a quiet room. Measured on the bench, a Pt1000 moved
   one digit every 75 minutes or so and sat perfectly still in between, which any
   plausible timeout reads as a dead channel. A false fault takes a WORKING sensor
   out of Home Assistant, which is worse than the case it was guarding against -
   and that case, an open circuit parked at an end of scale, is caught on the
   first scan by PlausibleMin/PlausibleMax anyway. *)
Fault := NOT Valid;

(* Self-restarting, so the heartbeat is a floor on how often the value is
   published rather than a timer anything has to remember to reset. *)
fbHeartbeat(IN := NOT fbHeartbeat.Q, PT := HeartbeatInterval);

(* --- publishing --------------------------------------------------------------
   Three reasons to publish and no others: the channel word changed, the heartbeat
   elapsed, or this is the first reading.

   There was a PublishDeadband input here, defaulting to 0.2 C, on the reasoning
   that an RTD's last digit dithers continuously and nobody wants that in their
   history. This bench measured the opposite - one digit every 75 minutes or so,
   dead still in between - so on a quiet channel it suppressed nothing, and it is
   gone. Every change is published, which is what setting it to zero always did.

   While the value is out of range nothing is published, deliberately: Temperature
   holds the last trustworthy reading, and the discovery config's expire_after lets
   Home Assistant retire the entity on its own if the silence lasts - a truer signal
   than publishing a made-up number, or the module's fault code dressed up as a
   temperature. *)
IF bInitMqttDone AND Valid THEN
	IF NOT bPublishedValid
		OR fbHeartbeat.Q
		OR (iCorrectedRaw <> iPublishedRaw)
	THEN
		(* Formatted from the integer rather than through REAL_TO_STRING, which
		   would publish 21.299999 for a channel reading 213. One decimal is all
		   the module has, and all anyone should be told it has. *)
		iWhole := iCorrectedRaw / 10;
		iTenth := ABS(iCorrectedRaw MOD 10);
		sPayload := INT_TO_STRING(iWhole);
		IF (Raw < 0) AND (iWhole = 0) THEN
			sPayload := CONCAT('-', sPayload);
		END_IF
		sPayload := CONCAT(sPayload, '.');
		sPayload := CONCAT(sPayload, INT_TO_STRING(iTenth));

		pMqttPublishQueue^.AddMessage(
			Payload := sPayload,
			Topic := CONCAT(THIS^.sMQTTPublishTopic, '/TEMP'),
			Qos := MQTT.QoS.ExactlyOnce,
			MqttRetain := TRUE);

		iPublishedRaw := iCorrectedRaw;
		bPublishedValid := TRUE;
	END_IF
END_IF

(* --- available, or not -------------------------------------------------------
   Published on change, both ways, plus once at startup - and that startup
   publish is not optional: Home Assistant treats a missing availability payload
   as unavailable, so an entity whose topic has never been written stays greyed
   out however healthy the channel is.

   This is the whole fault surface. There is no separate problem entity to go
   looking for: a channel that cannot be trusted greys out the temperature where
   somebody is already reading it. The value itself keeps being published while
   that happens, so a stuck channel's number is still on the broker for anyone
   who wants to judge it - it is just no longer presented as a measurement.

   The payloads come from GVL_MQTT rather than being spelled here, because they
   have to match the pl_avail / pl_not_avail that the discovery device published
   in the config, and that is where those come from. *)
fbFaultEdge(CLK := Fault);
fbHealEdge(CLK := Fault);

IF bInitMqttDone AND (bStartup OR fbFaultEdge.Q OR fbHealEdge.Q) THEN
	IF Fault THEN
		sPayload := GVL_MQTT.MqttAvailabilityOfflinePayload;
	ELSE
		sPayload := GVL_MQTT.MqttAvailabilityOnlinePayload;
	END_IF
	pMqttPublishQueue^.AddMessage(
		Payload := sPayload,
		Topic := CONCAT(THIS^.sMQTTPublishTopic, '/availability'),
		Qos := MQTT.QoS.ExactlyOnce,
		MqttRetain := TRUE);
	bStartup := FALSE;
END_IF

          

(* Publishes the Home Assistant MQTT discovery configs - a temperature sensor and a diagnostic fault flag - so both entities are created automatically. Call once at startup, after InitMqtt. *)
METHOD InitMqttDiscovery
  VAR_INPUT
    Device : POINTER TO FB_PLC_MQTT_DISCOVERY_DEVICE;  (* Pointer to the discovery device this entity belongs to, normally GVL_MQTT.PLC_Device. An RTD channel is part of the PLC rather than a device of its own. *)
    Name : STRING(255);  (* Name of the entity in Home Assistant. The self-wiring prologue passes FriendlyName. *)
    overruleId : STRING(255) := '';  (* Overrides the generated entity id. Leave empty to derive it from the function block name. *)
  END_VAR
  VAR
    id : STRING(255);
  END_VAR
                  IF bInitMqttDone AND NOT bInitMqttDiscoveryDone THEN

	id := SUPER^.ResolveEntityId(overruleId);

	(* One entity, and it goes unavailable when the reading cannot be trusted.

	   AvailabilityTopic overrides this entity's second availability topic, and
	   avty_mode is 'all', so Home Assistant shows the sensor only while the PLC
	   says online AND this channel says online. A fault therefore greys out the
	   temperature where somebody is already looking at it, rather than raising a
	   separate problem entity somewhere else to be noticed.

	   expire_after stays, at three heartbeats, as a backstop for the one case an
	   availability topic cannot cover: a PLC that stops publishing without
	   getting the chance to say so.

	   state_class measurement, so Home Assistant keeps long-term statistics -
	   unlike a distance, a temperature is exactly the kind of thing worth
	   graphing a mean of. *)
	Device^.CreateSensorEntity(
		Name := Name,
		Id := id,
		StateTopic := CONCAT(THIS^.sMQTTPublishTopic, '/TEMP'),
		ExpiryAfter := UDINT_TO_INT(TIME_TO_UDINT(HeartbeatInterval) * 3 / 1000),
		DeviceClass := 'temperature',
		UnitOfMeasurement := '°C',
		StateClass := 'measurement',
		AvailabilityTopic := CONCAT(THIS^.sMQTTPublishTopic, '/availability'));

	bInitMqttDiscoveryDone := TRUE;
END_IF
                
END_METHOD

(* Enables MQTT on the function block. Call once at startup. Not needed when FriendlyName is set at the declaration: the block then wires itself. *)
METHOD InitMqtt
  VAR_INPUT
    MQTTPublishPrefix : POINTER TO STRING;  (* Pointer to the MQTT publish prefix used for this block. The function block name is appended automatically. *)
    pMqttPublishQueue : POINTER TO FB_MQTT_PUBLISH_QUEUE;  (* Pointer to the shared MQTT queue that carries messages to the broker. *)
  END_VAR
                  SUPER^._sInstancePath := THIS^.sInstancePath; // Due to reflection its location is important

(*pass trough*)
THIS^.pMqttPublishQueue := pMqttPublishQueue;
THIS^.psMqttPublishTopicPrefix := MQTTPublishPrefix;
SUPER^.InitBaseMqtt();
                
END_METHOD
END_FUNCTION_BLOCK

{attribute 'reflection'}
FUNCTION_BLOCK FB_OUTPUT_BINARY_MQTT EXTENDS FB_MQTT_BASE IMPLEMENTS MQTT.MQTT_SUBSCRIBE_CALLBACK
  VAR_OUTPUT
    OUT : BOOL;
  END_VAR
  VAR
    {attribute 'noinit'}
    {attribute 'instance-path'}
    sInstancePath : STRING(GVL_MQTT.MQTT_TOPIC_LEN);  (* Refelection: object's full instance name *)
    bStartup : BOOL := TRUE;
  END_VAR
  VAR PERSISTENT
    bPreviousState : BOOL;  (* To retain output state through powercycles *)
  END_VAR
  VAR_INPUT
    PRIO_HIGH : BOOL := FALSE;
    PRIO_LOW : BOOL := FALSE;
    TOGGLE : BOOL := FALSE;
  END_VAR

            (* --- self-wiring prologue ----------------------------------------------------
   Makes the InitMqtt and InitMqttDiscovery* calls optional. Set FriendlyName at
   the declaration site and this block wires itself from GVL_MQTT on its
   first cyclic call, then announces itself to Home Assistant.

   Deliberately in the body rather than in FB_init: it dereferences GVL members
   and reads the reflection instance path, and doing that during initialisation
   would rely on an ordering nothing enforces and the compiler cannot check. The
   body is the same lifecycle phase the init actions used, so this is not merely
   safe, it is the phase that already works today.

   The wiring calls this block's own unmodified InitMqtt / InitMqttDiscovery*
   methods, so anything published - topics and discovery JSON alike - is produced
   by exactly the code that produces it today. Only the trigger moved.

   Dormant while FriendlyName is empty, so existing projects and existing call
   sites keep working untouched.

   A block wired this way MUST be called cyclically. An instance whose body never
   runs is now unwired and absent from Home Assistant, where the init action used
   to wire it regardless. Nothing warns about that.  *)
IF FriendlyName <> '' THEN

	IF NOT bInitMqttDone THEN
		THIS^.InitMqtt(
			MQTTPublishPrefix := ADR(GVL_MQTT.MqttPubSwitchPrefix),
			MQTTSubscribePrefix := ADR(GVL_MQTT.MqttSubSwitchPrefix),
			pMqttPublishQueue := ADR(GVL_MQTT.fbMqttPublishQueue),
			pMqttCallbackCollector := ADR(GVL_MQTT.collector_FB_OUTPUT_SWITCH_MQTT));
	END_IF

	IF bInitMqttDone AND NOT bInitMqttDiscoveryDone THEN
		IF EntityType = E_MQTT_ENTITY.Light THEN
			THIS^.InitMqttDiscoveryAsLight(
				Device := ADR(GVL_MQTT.PLC_Device),
				Name := FriendlyName,
				RelayType := RelayType);
		ELSIF EntityType = E_MQTT_ENTITY.Lock THEN
			THIS^.InitMqttDiscoveryAsLock(
				Device := ADR(GVL_MQTT.PLC_Device),
				Name := FriendlyName,
				RelayType := RelayType);
		ELSIF EntityType = E_MQTT_ENTITY.Siren THEN
			THIS^.InitMqttDiscoveryAsSiren(
				Device := ADR(GVL_MQTT.PLC_Device),
				Name := FriendlyName,
				RelayType := RelayType);
		ELSIF EntityType = E_MQTT_ENTITY.Valve THEN
			THIS^.InitMqttDiscoveryAsValve(
				Device := ADR(GVL_MQTT.PLC_Device),
				Name := FriendlyName,
				RelayType := RelayType);
		ELSIF EntityType = E_MQTT_ENTITY.Fan THEN
			THIS^.InitMqttDiscoveryAsFan(
				Device := ADR(GVL_MQTT.PLC_Device),
				Name := FriendlyName,
				RelayType := RelayType);
		ELSE
			(* Default, and any platform this block cannot announce as. *)
			THIS^.InitMqttDiscoveryAsSwitch(
				Device := ADR(GVL_MQTT.PLC_Device),
				Name := FriendlyName,
				RelayType := RelayType);
		END_IF
	END_IF

END_IF

IF bStartup THEN
	OUT := bPreviousState;
END_IF

IF PRIO_HIGH THEN
	OUT:=TRUE;
ELSIF(PRIO_LOW AND NOT (PRIO_HIGH)) THEN
	OUT:= FALSE;
ELSIF bMqttHighRequest THEN
	OUT:= TRUE;
	bMqttHighRequest := FALSE;
	bMqttLowRequest := FALSE;
ELSIF bMqttLowRequest THEN
	OUT:= FALSE;
	bMqttHighRequest := FALSE;
	bMqttLowRequest := FALSE;
ELSIF(TOGGLE) THEN
	OUT:=NOT(OUT);
END_IF;

IF ((bPreviousState <> OUT) OR bStartup) AND bInitMqttDone THEN
	pMqttPublishQueue^.AddMessage(
		Payload := BOOL_TO_STRING(OUT),
		Topic := sMQTTPublishTopic,
		Qos := MQTT.QoS.ExactlyOnce,
		MqttRetain := TRUE
	);	
	bStartup:=FALSE;
END_IF	

bPreviousState := OUT;
          

METHOD InitMqttDiscoveryAsSiren
  VAR_INPUT
    Device : POINTER TO FB_PLC_MQTT_DISCOVERY_DEVICE;
    Name : STRING(255);
    overruleId : STRING(255) := '';
    RelayType : E_RELAY_TYPE := E_RELAY_TYPE.NO;  (* NO (default) or NC. Swaps the payload pair so the entity reports the state of the load, not of the coil. *)
  END_VAR
  VAR
    id : STRING(255);
  END_VAR
                  IF bInitMqttDone AND NOT bInitMqttDiscoveryDone THEN
	
	id := SUPER^.ResolveEntityId(overruleId);
	
	Device^.CreateSirenEntity(
			Name := name,
			Id := id,
			CommandTopic := THIS^.sMQTTSubscribeTopic,
			PayloadOn := BOOL_TO_STRING(RelayType = E_RELAY_TYPE.NO),
			PayloadOff := BOOL_TO_STRING(RelayType = E_RELAY_TYPE.NC),
			StateTopic := THIS^.sMQTTPublishTopic,
			StateOnPayload := BOOL_TO_STRING(RelayType = E_RELAY_TYPE.NO),
			StateOffPayload := BOOL_TO_STRING(RelayType = E_RELAY_TYPE.NC)
		);


	bInitMqttDiscoveryDone := TRUE;
END_IF		
                
END_METHOD

METHOD InitMqttDiscoveryAsLock
  VAR_INPUT
    Device : POINTER TO FB_PLC_MQTT_DISCOVERY_DEVICE;
    Name : STRING(255);
    overruleId : STRING(255) := '';
    RelayType : E_RELAY_TYPE := E_RELAY_TYPE.NO;  (* NO (default) or NC. Swaps the payload pair so the entity reports the state of the load, not of the coil. *)
  END_VAR
  VAR
    id : STRING(255);
  END_VAR
                  IF bInitMqttDone AND NOT bInitMqttDiscoveryDone THEN
	
	id := SUPER^.ResolveEntityId(overruleId);
	
	Device^.CreateLockEntity(
		Name := name,
		Id := id,
		CommandTopic := THIS^.sMQTTSubscribeTopic,
		PayloadLock := BOOL_TO_STRING(RelayType = E_RELAY_TYPE.NO),
		PayloadUnlock := BOOL_TO_STRING(RelayType = E_RELAY_TYPE.NC),
		StateTopic := THIS^.sMQTTPublishTopic,
		StateUnlocked := BOOL_TO_STRING(RelayType = E_RELAY_TYPE.NC),
		StateLocked := BOOL_TO_STRING(RelayType = E_RELAY_TYPE.NO));

	bInitMqttDiscoveryDone := TRUE;
END_IF		
                
END_METHOD

METHOD InitMqttDiscoveryAsLight
  VAR_INPUT
    Device : POINTER TO FB_PLC_MQTT_DISCOVERY_DEVICE;
    Name : STRING(255);
    overruleId : STRING(255) := '';
    RelayType : E_RELAY_TYPE := E_RELAY_TYPE.NO;  (* NO (default) or NC. Swaps the payload pair so the entity reports the state of the load, not of the coil. *)
  END_VAR
  VAR
    id : STRING(255);
  END_VAR
                  IF bInitMqttDone AND NOT bInitMqttDiscoveryDone THEN
	
	id := SUPER^.ResolveEntityId(overruleId);
	
	Device^.CreateLightEntity(
			Name := name,
			Id := id,
			CommandTopic := THIS^.sMQTTSubscribeTopic,
			PayloadOn := BOOL_TO_STRING(RelayType = E_RELAY_TYPE.NO),
			PayloadOff := BOOL_TO_STRING(RelayType = E_RELAY_TYPE.NC),
			StateTopic := THIS^.sMQTTPublishTopic);

	bInitMqttDiscoveryDone := TRUE;
END_IF		
                
END_METHOD

METHOD InitMqttDiscoveryAsSwitch
  VAR_INPUT
    Device : POINTER TO FB_PLC_MQTT_DISCOVERY_DEVICE;
    Name : STRING(255);
    DeviceClass : STRING(100) := 'outlet';
    overruleId : STRING(255) := '';
    RelayType : E_RELAY_TYPE := E_RELAY_TYPE.NO;  (* NO (default) or NC. Swaps the payload pair so the entity reports the state of the load, not of the coil. *)
  END_VAR
  VAR
    id : STRING(255);
  END_VAR
                  IF bInitMqttDone AND NOT bInitMqttDiscoveryDone THEN
	
	id := SUPER^.ResolveEntityId(overruleId);
	
	Device^.CreateSwitchEntity(
			Name := name,
			Id := id,
			CommandTopic := THIS^.sMQTTSubscribeTopic,
			PayloadOn := BOOL_TO_STRING(RelayType = E_RELAY_TYPE.NO),
			PayloadOff := BOOL_TO_STRING(RelayType = E_RELAY_TYPE.NC),
			StateTopic := THIS^.sMQTTPublishTopic,
			StateOnPayload := BOOL_TO_STRING(RelayType = E_RELAY_TYPE.NO),
			StateOffPayload := BOOL_TO_STRING(RelayType = E_RELAY_TYPE.NC),
			DeviceClass := DeviceClass);
	
	bInitMqttDiscoveryDone := TRUE;
END_IF		
                
END_METHOD

METHOD PublishReceived : BOOL
  VAR_INPUT
    Data : MQTT.CALLBACK_DATA;  (* Collection of recived Data *)
  END_VAR
                  //first check if Mqtt is initialized, otherwise do nothing
IF NOT(bInitMqttDone) THEN
	//mark the interface call from the collector as done
	PublishReceived := TRUE;
//check if the packet is for this FB
ELSIF CommonTypesAndFunctions.StrEquals(str1:= ADR(sMQTTSubscribeTopic), str2:= Data.TopicOut) THEN
	//mark the interface call from the collector as done
	PublishReceived := TRUE;
	//now process the data
	IF CommonTypesAndFunctions.StrEquals(str1:= Data.PayloadString, str2:= ADR('TRUE')) THEN
		bMqttHighRequest := TRUE;
	ELSIF CommonTypesAndFunctions.StrEquals(str1:= Data.PayloadString, str2:= ADR('FALSE')) THEN
		bMqttLowRequest := TRUE;
	// Siren sends out a JSON
	ELSIF FIND(Data.PayloadString^, 'TRUE') > 0 THEN
		bMqttHighRequest := TRUE;
	ELSIF FIND(Data.PayloadString^, 'FALSE') > 0 THEN
		bMqttLowRequest := TRUE;
	END_IF
END_IF 
                
END_METHOD

METHOD InitMqtt
  VAR_INPUT
    MQTTPublishPrefix : POINTER TO STRING;
    MQTTSubscribePrefix : POINTER TO STRING;
    pMqttPublishQueue : POINTER TO FB_MQTT_PUBLISH_QUEUE;
    pMqttCallbackCollector : POINTER TO MQTT.CallbackCollector;
  END_VAR
                  SUPER^._sInstancePath := THIS^.sInstancePath; // Due to reflection its location is important

(*pass trough*)
THIS^.pMqttPublishQueue := pMqttPublishQueue;
THIS^.psMqttPublishTopicPrefix:=MQTTPublishPrefix;
THIS^.psMqttSubscribeTopicPrefix:=MQTTSubscribePrefix;
THIS^.pMqttPublishQueue:=pMqttPublishQueue;

SUPER^.InitBaseMqtt();
pMqttCallbackCollector^.put(instance:= THIS^); // register the FB agains the collector so mqtt events can be received


                
END_METHOD

METHOD InitMqttDiscoveryAsValve
  VAR_INPUT
    Device : POINTER TO FB_PLC_MQTT_DISCOVERY_DEVICE;
    Name : STRING(255);
    DeviceClass : STRING(100) := 'water';  (* water or gas *)
    overruleId : STRING(255) := '';
    RelayType : E_RELAY_TYPE := E_RELAY_TYPE.NO;  (* NO (default) or NC. Swaps the payload pair so the entity reports the state of the load, not of the coil. *)
  END_VAR
  VAR
    id : STRING(255);
  END_VAR
                  IF bInitMqttDone AND NOT bInitMqttDiscoveryDone THEN
	
	id := SUPER^.ResolveEntityId(overruleId);
	
	Device^.CreateValveEntity(
			Name := name,
			Id := id,
			CommandTopic := THIS^.sMQTTSubscribeTopic,
			PayloadOpen := BOOL_TO_STRING(RelayType = E_RELAY_TYPE.NO),
			PayloadClosed := BOOL_TO_STRING(RelayType = E_RELAY_TYPE.NC),
			StateTopic := THIS^.sMQTTPublishTopic,
			StateOpen := BOOL_TO_STRING(RelayType = E_RELAY_TYPE.NO),
			StateClosed := BOOL_TO_STRING(RelayType = E_RELAY_TYPE.NC),
			Deviceclass := DeviceClass);

	bInitMqttDiscoveryDone := TRUE;
END_IF		
                
END_METHOD

METHOD InitMqttDiscoveryAsFan
  VAR_INPUT
    Device : POINTER TO FB_PLC_MQTT_DISCOVERY_DEVICE;
    Name : STRING(255);
    overruleId : STRING(255) := '';
    RelayType : E_RELAY_TYPE := E_RELAY_TYPE.NO;  (* NO (default) or NC. Swaps the payload pair so the entity reports the state of the load, not of the coil. *)
  END_VAR
  VAR
    id : STRING(255);
  END_VAR
                  IF bInitMqttDone AND NOT bInitMqttDiscoveryDone THEN

	id := SUPER^.ResolveEntityId(overruleId);

	(* An on/off fan: no percentage or oscillation topics, because a binary output
	   has no speed to report. A E_DIMMER-backed fan would pass those. *)
	Device^.CreateFanEntity(
			Name := name,
			Id := id,
			CommandTopic := THIS^.sMQTTSubscribeTopic,
			PayloadOn := BOOL_TO_STRING(RelayType = E_RELAY_TYPE.NO),
			PayloadOff := BOOL_TO_STRING(RelayType = E_RELAY_TYPE.NC),
			StateTopic := THIS^.sMQTTPublishTopic);

	bInitMqttDiscoveryDone := TRUE;
END_IF
                
END_METHOD
END_FUNCTION_BLOCK

{attribute 'reflection'}
FUNCTION_BLOCK FB_OUTPUT_BISTABLE_MQTT EXTENDS FB_MQTT_BASE IMPLEMENTS MQTT.MQTT_SUBSCRIBE_CALLBACK
  VAR_OUTPUT
    OUT : BOOL;
  END_VAR
  VAR
    {attribute 'noinit'}
    {attribute 'instance-path'}
    sInstancePath : STRING(GVL_MQTT.MQTT_TOPIC_LEN);  (* Refelection: object's full instance name *)
    bStartup : BOOL := TRUE;
    bPreviousFeedback : BOOL;
    fbHoldTimer : TOF;
    T_hold : TIME := TIME#1s0ms;
    bPulseTrigger : BOOL := FALSE;
  END_VAR
  VAR_INPUT
    PRIO_HIGH : BOOL := FALSE;
    PRIO_LOW : BOOL := FALSE;
    TOGGLE : BOOL := FALSE;
    FEEDBACK : BOOL := FALSE;
  END_VAR

            (* --- self-wiring prologue ----------------------------------------------------
   Makes the InitMqtt and InitMqttDiscovery* calls optional. Set FriendlyName at
   the declaration site and this block wires itself from GVL_MQTT on its
   first cyclic call, then announces itself to Home Assistant.

   Deliberately in the body rather than in FB_init: it dereferences GVL members
   and reads the reflection instance path, and doing that during initialisation
   would rely on an ordering nothing enforces and the compiler cannot check. The
   body is the same lifecycle phase the init actions used, so this is not merely
   safe, it is the phase that already works today.

   The wiring calls this block's own unmodified InitMqtt / InitMqttDiscovery*
   methods, so anything published - topics and discovery JSON alike - is produced
   by exactly the code that produces it today. Only the trigger moved.

   Dormant while FriendlyName is empty, so existing projects and existing call
   sites keep working untouched.

   A block wired this way MUST be called cyclically. An instance whose body never
   runs is now unwired and absent from Home Assistant, where the init action used
   to wire it regardless. Nothing warns about that.  *)
IF FriendlyName <> '' THEN

	IF NOT bInitMqttDone THEN
		THIS^.InitMqtt(
			MQTTPublishPrefix := ADR(GVL_MQTT.MqttPubSwitchPrefix),
			MQTTSubscribePrefix := ADR(GVL_MQTT.MqttSubSwitchPrefix),
			pMqttPublishQueue := ADR(GVL_MQTT.fbMqttPublishQueue),
			pMqttCallbackCollector := ADR(GVL_MQTT.collector_FB_OUTPUT_SWITCH_MQTT));
	END_IF

	IF bInitMqttDone AND NOT bInitMqttDiscoveryDone THEN
		IF EntityType = E_MQTT_ENTITY.Light THEN
			THIS^.InitMqttDiscoveryAsLight(
				Device := ADR(GVL_MQTT.PLC_Device),
				Name := FriendlyName,
				RelayType := RelayType);
		ELSIF EntityType = E_MQTT_ENTITY.Lock THEN
			THIS^.InitMqttDiscoveryAsLock(
				Device := ADR(GVL_MQTT.PLC_Device),
				Name := FriendlyName,
				RelayType := RelayType);
		ELSIF EntityType = E_MQTT_ENTITY.Siren THEN
			THIS^.InitMqttDiscoveryAsSiren(
				Device := ADR(GVL_MQTT.PLC_Device),
				Name := FriendlyName,
				RelayType := RelayType);
		ELSIF EntityType = E_MQTT_ENTITY.Fan THEN
			THIS^.InitMqttDiscoveryAsFan(
				Device := ADR(GVL_MQTT.PLC_Device),
				Name := FriendlyName,
				RelayType := RelayType);
		ELSE
			(* Default, and any platform this block cannot announce as. *)
			THIS^.InitMqttDiscoveryAsSwitch(
				Device := ADR(GVL_MQTT.PLC_Device),
				Name := FriendlyName,
				RelayType := RelayType);
		END_IF
	END_IF

END_IF

fbHoldTimer(PT:= T_hold);

IF PRIO_HIGH THEN
	IF NOT FEEDBACK THEN
		bPulseTrigger:=TRUE;
	END_IF
ELSIF(PRIO_LOW AND NOT (PRIO_HIGH)) THEN
	IF FEEDBACK THEN		
		bPulseTrigger:=TRUE;
	END_IF
	OUT:= FALSE;
ELSIF bMqttHighRequest THEN
	IF NOT FEEDBACK THEN		
		bPulseTrigger:=TRUE;
	END_IF
	bMqttHighRequest := FALSE;
	bMqttLowRequest := FALSE;
ELSIF bMqttLowRequest THEN
	IF FEEDBACK THEN		
		bPulseTrigger:=TRUE;
	END_IF
	bMqttHighRequest := FALSE;
	bMqttLowRequest := FALSE;
ELSIF(TOGGLE) THEN	
	bPulseTrigger:=TRUE;
END_IF;

IF ((bPreviousFeedback <> FEEDBACK) OR bStartup) AND bInitMqttDone THEN
	pMqttPublishQueue^.AddMessage(
		Payload := BOOL_TO_STRING(FEEDBACK),
		Topic := CONCAT(psMqttPublishTopicPrefix^, MqttPublishTopicSuffix),
		Qos := MQTT.QoS.ExactlyOnce,
		MqttRetain := TRUE
	);	
	bStartup:=FALSE;
END_IF	

bPreviousFeedback := FEEDBACK;
fbHoldTimer.IN	 := bPulseTrigger;
OUT := fbHoldTimer.Q;

bPulseTrigger:=FALSE;
          

METHOD InitMqttDiscoveryAsLight
  VAR_INPUT
    Device : POINTER TO FB_PLC_MQTT_DISCOVERY_DEVICE;
    Name : STRING(255);
    overruleId : STRING(255) := '';
    RelayType : E_RELAY_TYPE := E_RELAY_TYPE.NO;  (* NO (default) or NC. Swaps the payload pair so the entity reports the state of the load, not of the coil. *)
  END_VAR
  VAR
    id : STRING(255);
  END_VAR
                  IF bInitMqttDone AND NOT bInitMqttDiscoveryDone THEN
	
	id := SUPER^.ResolveEntityId(overruleId);
	
	Device^.CreateLightEntity(
			Name := name,
			Id := id,
			CommandTopic := THIS^.sMQTTSubscribeTopic,
			PayloadOn := BOOL_TO_STRING(RelayType = E_RELAY_TYPE.NO),
			PayloadOff := BOOL_TO_STRING(RelayType = E_RELAY_TYPE.NC),
			StateTopic := THIS^.sMQTTPublishTopic);

	bInitMqttDiscoveryDone := TRUE;
END_IF		
                
END_METHOD

METHOD InitMqttDiscoveryAsLock
  VAR_INPUT
    Device : POINTER TO FB_PLC_MQTT_DISCOVERY_DEVICE;
    Name : STRING(255);
    overruleId : STRING(255) := '';
    RelayType : E_RELAY_TYPE := E_RELAY_TYPE.NO;  (* NO (default) or NC. Swaps the payload pair so the entity reports the state of the load, not of the coil. *)
  END_VAR
  VAR
    id : STRING(255);
  END_VAR
                  IF bInitMqttDone AND NOT bInitMqttDiscoveryDone THEN
	
	id := SUPER^.ResolveEntityId(overruleId);
	
	Device^.CreateLockEntity(
		Name := name,
		Id := id,
		CommandTopic := THIS^.sMQTTSubscribeTopic,
		PayloadLock := BOOL_TO_STRING(RelayType = E_RELAY_TYPE.NO),
		PayloadUnlock := BOOL_TO_STRING(RelayType = E_RELAY_TYPE.NC),
		StateTopic := THIS^.sMQTTPublishTopic,
		StateUnlocked := BOOL_TO_STRING(RelayType = E_RELAY_TYPE.NC),
		StateLocked := BOOL_TO_STRING(RelayType = E_RELAY_TYPE.NO));

	bInitMqttDiscoveryDone := TRUE;
END_IF		
                
END_METHOD

METHOD InitMqttDiscoveryAsSiren
  VAR_INPUT
    Device : POINTER TO FB_PLC_MQTT_DISCOVERY_DEVICE;
    Name : STRING(255);
    overruleId : STRING(255) := '';
    RelayType : E_RELAY_TYPE := E_RELAY_TYPE.NO;  (* NO (default) or NC. Swaps the payload pair so the entity reports the state of the load, not of the coil. *)
  END_VAR
  VAR
    id : STRING(255);
  END_VAR
                  IF bInitMqttDone AND NOT bInitMqttDiscoveryDone THEN
	
	id := SUPER^.ResolveEntityId(overruleId);
	
	Device^.CreateSirenEntity(
			Name := name,
			Id := id,
			CommandTopic := THIS^.sMQTTSubscribeTopic,
			PayloadOn := BOOL_TO_STRING(RelayType = E_RELAY_TYPE.NO),
			PayloadOff := BOOL_TO_STRING(RelayType = E_RELAY_TYPE.NC),
			StateTopic := THIS^.sMQTTPublishTopic,
			StateOnPayload := BOOL_TO_STRING(RelayType = E_RELAY_TYPE.NO),
			StateOffPayload := BOOL_TO_STRING(RelayType = E_RELAY_TYPE.NC)
		);

	bInitMqttDiscoveryDone := TRUE;
END_IF		
                
END_METHOD

METHOD InitMqtt
  VAR_INPUT
    MQTTPublishPrefix : POINTER TO STRING;
    MQTTSubscribePrefix : POINTER TO STRING;
    pMqttPublishQueue : POINTER TO FB_MQTT_PUBLISH_QUEUE;
    pMqttCallbackCollector : POINTER TO MQTT.CallbackCollector;
  END_VAR
                  SUPER^._sInstancePath := THIS^.sInstancePath; // Due to reflection its location is important

(*pass trough*)
THIS^.pMqttPublishQueue := pMqttPublishQueue;
THIS^.psMqttPublishTopicPrefix:=MQTTPublishPrefix;
THIS^.psMqttSubscribeTopicPrefix:=MQTTSubscribePrefix;
THIS^.pMqttPublishQueue:=pMqttPublishQueue;



SUPER^.InitBaseMqtt();
pMqttCallbackCollector^.put(instance:= THIS^); // register the FB agains the collector so mqtt events can be received


                
END_METHOD

METHOD PublishReceived : BOOL
  VAR_INPUT
    Data : MQTT.CALLBACK_DATA;  (* Collection of recived Data *)
  END_VAR
                  //first check if Mqtt is initialized, otherwise do nothing
IF NOT(bInitMqttDone) THEN
	//mark the interface call from the collector as done
	PublishReceived := TRUE;
//check if the packet is for this FB
ELSIF CommonTypesAndFunctions.StrEquals(str1:= ADR(sMQTTSubscribeTopic), str2:= Data.TopicOut) THEN
	//mark the interface call from the collector as done
	PublishReceived := TRUE;
	//now process the data
	IF CommonTypesAndFunctions.StrEquals(str1:= Data.PayloadString, str2:= ADR('TRUE')) THEN
		bMqttHighRequest := TRUE;
	ELSIF CommonTypesAndFunctions.StrEquals(str1:= Data.PayloadString, str2:= ADR('FALSE')) THEN
		bMqttLowRequest := TRUE;
	// Siren sends out a JSON
	ELSIF FIND(Data.PayloadString^, 'TRUE') > 0 THEN
		bMqttHighRequest := TRUE;
	ELSIF FIND(Data.PayloadString^, 'FALSE') > 0 THEN
		bMqttLowRequest := TRUE;
	END_IF
END_IF 
                
END_METHOD

METHOD ConfigureFunctionBlock
  VAR_INPUT
    T_hold : TIME;  (* Default value for click mode, can be overwritten by method call *)
  END_VAR
                  THIS^.T_hold:=T_hold;
                
END_METHOD

METHOD InitMqttDiscoveryAsSwitch
  VAR_INPUT
    Device : POINTER TO FB_PLC_MQTT_DISCOVERY_DEVICE;
    Name : STRING(255);
    DeviceClass : STRING(100) := 'outlet';
    overruleId : STRING(255) := '';
    RelayType : E_RELAY_TYPE := E_RELAY_TYPE.NO;  (* NO (default) or NC. Swaps the payload pair so the entity reports the state of the load, not of the coil. *)
  END_VAR
  VAR
    id : STRING(255);
  END_VAR
                  IF bInitMqttDone AND NOT bInitMqttDiscoveryDone THEN
	
	id := SUPER^.ResolveEntityId(overruleId);
	
	Device^.CreateSwitchEntity(
			Name := name,
			Id := id,
			CommandTopic := THIS^.sMQTTSubscribeTopic,
			PayloadOn := BOOL_TO_STRING(RelayType = E_RELAY_TYPE.NO),
			PayloadOff := BOOL_TO_STRING(RelayType = E_RELAY_TYPE.NC),
			StateTopic := THIS^.sMQTTPublishTopic,
			StateOnPayload := BOOL_TO_STRING(RelayType = E_RELAY_TYPE.NO),
			StateOffPayload := BOOL_TO_STRING(RelayType = E_RELAY_TYPE.NC),
			DeviceClass := DeviceClass);
	
	bInitMqttDiscoveryDone := TRUE;
END_IF		
                
END_METHOD

METHOD InitMqttDiscoveryAsFan
  VAR_INPUT
    Device : POINTER TO FB_PLC_MQTT_DISCOVERY_DEVICE;
    Name : STRING(255);
    overruleId : STRING(255) := '';
    RelayType : E_RELAY_TYPE := E_RELAY_TYPE.NO;  (* NO (default) or NC. Swaps the payload pair so the entity reports the state of the load, not of the coil. *)
  END_VAR
  VAR
    id : STRING(255);
  END_VAR
                  IF bInitMqttDone AND NOT bInitMqttDiscoveryDone THEN

	id := SUPER^.ResolveEntityId(overruleId);

	(* An on/off fan: no percentage or oscillation topics, because a binary output
	   has no speed to report. A E_DIMMER-backed fan would pass those. *)
	Device^.CreateFanEntity(
			Name := name,
			Id := id,
			CommandTopic := THIS^.sMQTTSubscribeTopic,
			PayloadOn := BOOL_TO_STRING(RelayType = E_RELAY_TYPE.NO),
			PayloadOff := BOOL_TO_STRING(RelayType = E_RELAY_TYPE.NC),
			StateTopic := THIS^.sMQTTPublishTopic);

	bInitMqttDiscoveryDone := TRUE;
END_IF
                
END_METHOD
END_FUNCTION_BLOCK

{attribute 'reflection'}
FUNCTION_BLOCK FB_OUTPUT_COVER_MQTT EXTENDS FB_MQTT_BASE IMPLEMENTS MQTT.MQTT_SUBSCRIBE_CALLBACK
  VAR_OUTPUT
    MU : BOOL;
    MD : BOOL;
  END_VAR
  VAR
    {attribute 'noinit'}
    {attribute 'instance-path'}
    sInstancePath : STRING(GVL_MQTT.MQTT_TOPIC_LEN);  (* object's full instance name *)
    fbLock : OSCAT_BASIC.INTERLOCK;
    fbCoverStateTimer : TOF;
    bInternalUp : BOOL;
    bInternalDown : BOOL;
    bMqttRequestStop : BOOL;
    bMqttRequestOpen : BOOL;
    bMqttRequestClose : BOOL;
    fbMuRTrigger : Standard.R_TRIG;
    fbMdRTrigger : Standard.R_TRIG;
    fbMuFTrigger : Standard.F_TRIG;
    fbMdFTrigger : Standard.F_TRIG;
    bStartup : BOOL := TRUE;  (* Drives a single state publish at boot, matching every sibling block. *)
    T_LOCKOUT : TIME := TIME#1s0ms;  (* Delay between a change of direction, so the motor is never driven both ways at once. Set once by FB_init at the instance declaration. *)
    T_UD : TIME := TIME#10s0ms;  (* Run time to move the cover completely up or down. Set once by FB_init at the instance declaration. *)
  END_VAR
  VAR PERSISTENT
    bInternalDir : BOOL;  (* down = false, up = true *)
  END_VAR
  VAR_INPUT
    TOGGLE : BOOL;
    PRIO_LOCK : BOOL;
    PRIO_UP : BOOL;
    PRIO_DN : BOOL;
  END_VAR

            (* --- self-wiring prologue ----------------------------------------------------
   Makes the InitMqtt and InitMqttDiscovery* calls optional. Set FriendlyName at
   the declaration site and this block wires itself from GVL_MQTT on its
   first cyclic call, then announces itself to Home Assistant.

   Deliberately in the body rather than in FB_init: it dereferences GVL members
   and reads the reflection instance path, and doing that during initialisation
   would rely on an ordering nothing enforces and the compiler cannot check. The
   body is the same lifecycle phase the init actions used, so this is not merely
   safe, it is the phase that already works today.

   The wiring calls this block's own unmodified InitMqtt / InitMqttDiscovery*
   methods, so anything published - topics and discovery JSON alike - is produced
   by exactly the code that produces it today. Only the trigger moved.

   Dormant while FriendlyName is empty, so existing projects and existing call
   sites keep working untouched.

   A block wired this way MUST be called cyclically. An instance whose body never
   runs is now unwired and absent from Home Assistant, where the init action used
   to wire it regardless. Nothing warns about that.  *)
IF FriendlyName <> '' THEN

	IF NOT bInitMqttDone THEN
		THIS^.InitMqtt(
			MQTTPublishPrefix := ADR(GVL_MQTT.MqttPubCoverPrefix),
			MQTTSubscribePrefix := ADR(GVL_MQTT.MqttSubCoverPrefix),
			pMqttPublishQueue := ADR(GVL_MQTT.fbMqttPublishQueue),
			pMqttCallbackCollector := ADR(GVL_MQTT.collector_FB_OUTPUT_COVER_MQTT));
	END_IF

	IF bInitMqttDone AND NOT bInitMqttDiscoveryDone THEN
		THIS^.InitMqttDiscovery(
			Device := ADR(GVL_MQTT.PLC_Device),
			Name := FriendlyName);
	END_IF

END_IF

(* Run the timer to not power the motors for to long *)
fbCoverStateTimer(PT:=T_UD);
fbCoverStateTimer.IN:=FALSE;
fbMuRTrigger(CLK:=MU);
fbMdRTrigger(CLK:=MD);
fbMuFTrigger(CLK:=MU);
fbMdFTrigger(CLK:=MD);

(* Publish once at boot so the entity has a value before the first movement.
   Deliberately 'STOPPED' rather than a derived OPEN/CLOSED: bInternalDir is
   PERSISTENT and does carry the last direction, but its meaning is ambiguous -
   the declaration comment says "down = false, up = true" while the logic below
   sets bInternalDir := FALSE after a completed upward move. 'STOPPED' is an
   honest "position unknown", and a confidently wrong OPEN or CLOSED would
   mislead automations more than no position does. *)
IF bStartup AND bInitMqttDone THEN
	bStartup := FALSE;
	pMqttPublishQueue^.AddMessage(
		Payload := 'STOPPED',
		Topic := CONCAT(psMqttPublishTopicPrefix^, MqttPublishTopicSuffix),
		Qos := MQTT.QoS.ExactlyOnce,
		MqttRetain := TRUE
	);
END_IF

IF fbMuRTrigger.Q AND bInitMqttDone THEN
	pMqttPublishQueue^.AddMessage(
		Payload := 'OPENING',
		Topic := CONCAT(psMqttPublishTopicPrefix^, MqttPublishTopicSuffix),
		Qos := MQTT.QoS.ExactlyOnce,
		MqttRetain := TRUE
	);
END_IF

IF fbMdRTrigger.Q AND bInitMqttDone THEN
	pMqttPublishQueue^.AddMessage(
		Payload := 'CLOSING',
		Topic := CONCAT(psMqttPublishTopicPrefix^, MqttPublishTopicSuffix),
		Qos := MQTT.QoS.ExactlyOnce,
		MqttRetain := TRUE
	);
END_IF	

IF (fbMdFTrigger.Q OR fbMuFTrigger.Q) AND fbCoverStateTimer.Q AND bInitMqttDone THEN
	pMqttPublishQueue^.AddMessage(
		Payload := 'STOPPED',
		Topic := CONCAT(psMqttPublishTopicPrefix^, MqttPublishTopicSuffix),
		Qos := MQTT.QoS.ExactlyOnce,
		MqttRetain := TRUE
	);
END_IF	


IF (NOT(fbCoverStateTimer.Q) AND bInternalUp) AND bInitMqttDone THEN
	pMqttPublishQueue^.AddMessage(
		Payload := 'OPEN',
		Topic := CONCAT(psMqttPublishTopicPrefix^, MqttPublishTopicSuffix),
		Qos := MQTT.QoS.ExactlyOnce,
		MqttRetain := TRUE
	);
END_IF

IF (NOT(fbCoverStateTimer.Q) AND bInternalDown) AND bInitMqttDone THEN
	pMqttPublishQueue^.AddMessage(
		Payload := 'CLOSED',
		Topic := CONCAT(psMqttPublishTopicPrefix^, MqttPublishTopicSuffix),
		Qos := MQTT.QoS.ExactlyOnce,
		MqttRetain := TRUE
	);
END_IF


(* Check what to do *)
IF NOT(fbCoverStateTimer.Q) AND bInternalUp THEN // don't run the motors for to long, assume we've reached end and toggle dir
	bInternalUp := FALSE;
	bInternalDown := FALSE;
	bInternalDir := FALSE;
ELSIF NOT(fbCoverStateTimer.Q) AND bInternalDown THEN // don't run the motors for to long, assume we've reached end and toggle dir
	bInternalUp := FALSE;
	bInternalDown := FALSE;
	bInternalDir := TRUE;
ELSIF PRIO_LOCK THEN	
	bInternalUp := FALSE;
	bInternalDown := FALSE;
ELSIF PRIO_UP THEN	
	bInternalUp := TRUE;
	bInternalDown := FALSE;
	fbCoverStateTimer.IN:=TRUE;
ELSIF PRIO_DN THEN	
	bInternalUp := FALSE;
	bInternalDown := TRUE;
	fbCoverStateTimer.IN:=TRUE;
ELSIF TOGGLE AND (bInternalUp OR bInternalDown) THEN	// stop and toggle dir
	bInternalUp := FALSE;
	bInternalDown := FALSE;
	bInternalDir := NOT(bInternalDir);
ELSIF TOGGLE AND NOT(bInternalDir) THEN //move down
	bInternalUp := FALSE;
	bInternalDown := TRUE;
	fbCoverStateTimer.IN:=TRUE;
ELSIF TOGGLE AND bInternalDir THEN //move upwards
	bInternalUp := TRUE;
	bInternalDown := FALSE;	
	fbCoverStateTimer.IN:=TRUE;
ELSIF bMqttRequestStop THEN
	bInternalUp := FALSE;
	bInternalDown := FALSE;
	bMqttRequestStop := FALSE;
ELSIF bMqttRequestOpen THEN
	bInternalUp := TRUE;
	bInternalDown := FALSE;
	bMqttRequestOpen := FALSE;
	fbCoverStateTimer.IN:=TRUE;;
ELSIF bMqttRequestClose THEN
	bInternalUp := FALSE;
	bInternalDown := TRUE;
	bMqttRequestClose := FALSE;
	fbCoverStateTimer.IN:=TRUE;
END_IF

(* make sure only one motor is active at a given time *)
fbLock(i1 := bInternalUp, I2 := bInternalDown, TL := T_lockout);
MU := fbLock.Q1;
MD := fbLock.Q2;
          

METHOD InitMqttDiscovery
  VAR_INPUT
    Device : POINTER TO FB_PLC_MQTT_DISCOVERY_DEVICE;
    Name : STRING(255);
    overruleId : STRING(255) := '';
    DeviceClass : STRING(50) := 'shutter';
  END_VAR
  VAR
    id : STRING(255);
  END_VAR
                  IF bInitMqttDone AND NOT bInitMqttDiscoveryDone THEN
	
	id := SUPER^.ResolveEntityId(overruleId);
	
	Device^.CreateCoverEntity(
		Name := name,
		Id := id,
		CommandTopic := THIS^.sMQTTSubscribeTopic,
		PayloadOpen := 'OPEN',
		PayloadClose := 'CLOSE',
		PayloadStop := 'STOP',
		StateTopic := THIS^.sMQTTPublishTopic,
		StateOpen := 'OPEN',
		StateOpening := 'OPENING',
		StateClosed := 'CLOSED',
		StateClosing := 'CLOSING',
		StateStopped := 'STOPPED',
		DeviceClass := DeviceClass
	);

	bInitMqttDiscoveryDone := TRUE;
END_IF
                
END_METHOD

METHOD PublishReceived : BOOL
  VAR_INPUT
    Data : MQTT.CALLBACK_DATA;  (* Collection of recived Data *)
  END_VAR
                  //first check if Mqtt is initialized, otherwise do nothing
IF NOT(bInitMqttDone) THEN
	//mark the interface call from the collector as done
	PublishReceived := TRUE;
//check if the packet is for this FB
ELSIF CommonTypesAndFunctions.StrEquals(str1:= ADR(sMQTTSubscribeTopic), str2:= Data.TopicOut) THEN
	//mark the interface call from the collector as done
	PublishReceived := TRUE;
	//now process the data
	IF CommonTypesAndFunctions.StrEquals(str1:= Data.PayloadString, str2:= ADR('STOP')) THEN			
		THIS^.bMqttRequestStop:=TRUE;
	ELSIF CommonTypesAndFunctions.StrEquals(str1:= Data.PayloadString, str2:= ADR('OPEN')) THEN
		THIS^.bMqttRequestOpen:=TRUE;
	ELSIF CommonTypesAndFunctions.StrEquals(str1:= Data.PayloadString, str2:= ADR('CLOSE')) THEN
		THIS^.bMqttRequestClose:=TRUE;
	END_IF

END_IF
                
END_METHOD

METHOD InitMqtt
  VAR_INPUT
    MQTTPublishPrefix : POINTER TO STRING;
    MQTTSubscribePrefix : POINTER TO STRING;
    pMqttPublishQueue : POINTER TO FB_MQTT_PUBLISH_QUEUE;
    pMqttCallbackCollector : POINTER TO MQTT.CallbackCollector;
  END_VAR
                  SUPER^._sInstancePath := THIS^.sInstancePath; // Due to reflection its location is important

(*pass trough*)
THIS^.pMqttPublishQueue := pMqttPublishQueue;
THIS^.psMqttPublishTopicPrefix:=MQTTPublishPrefix;
THIS^.psMqttSubscribeTopicPrefix:=MQTTSubscribePrefix;

SUPER^.InitBaseMqtt();
pMqttCallbackCollector^.put(instance:= THIS^); // register the FB agains the collector so mqtt events can be received
                
END_METHOD

(* FB_Init is always available implicitly and it is used primarily for initialization. The return value is not evaluated. For a specific influence, you can also declare the methods explicitly and provide additional code there with the standard initialization code. You can evaluate the return value. *)
METHOD FB_init : BOOL
  VAR_INPUT
    bInitRetains : BOOL;  (* TRUE: the retain variables are initialized (reset warm / reset cold) *)
    bInCopyCode : BOOL;  (* TRUE: the instance will be copied to the copy code afterward (online change) *)
    T_LOCKOUT : TIME;  (* Delay between a change of direction. *)
    T_UD : TIME;  (* Run time to move the cover completely up or down. *)
  END_VAR
                  (* Cover timings, fixed for the life of the instance. Deliberately here rather
   than in a Configure method: these describe the motor and the shutter, so
   there is no scenario in which they should change while the PLC runs, and a
   runtime setter invited exactly the contradiction this block used to carry -
   two input_constant attributes alongside a method that assigned them anyway.

   Touches only non-persistent members. FB_init runs on every download and
   reset, so writing bInternalDir here would destroy the retained direction. *)
THIS^.T_LOCKOUT := T_LOCKOUT;
THIS^.T_UD := T_UD;

                
END_METHOD
END_FUNCTION_BLOCK

{attribute 'reflection'}
FUNCTION_BLOCK FB_OUTPUT_COVER_POSITION_MQTT EXTENDS FB_MQTT_BASE IMPLEMENTS MQTT.MQTT_SUBSCRIBE_CALLBACK
  VAR_INPUT
    UP : BOOL;  (* Manual up, e.g. straight from a pushbutton's long-press output. Held TRUE drives the motor up and releasing it stops and holds where it is, which is what a physical button should do - the position it was travelling to is abandoned rather than resumed. *)
    DN : BOOL;  (* Manual down, same contract as UP. Both at once is not a command and is ignored, because there is no sane guess to make. *)
    PRIO_LOCK : BOOL;  (* Nothing may drive the motor while this is TRUE - a wind alarm, a service switch, an open window contact. Commands are still accepted and still remembered; they simply do not move anything until it clears. *)
    T_TravelUp : TIME := TIME#20s0ms;  (* How long the cover takes to travel from fully closed to fully open, and back. These two are how the position is known at all: there is no encoder on a shutter motor, so run time is integrated against them. Measure them rather than guessing, and measure both - a shutter usually falls faster than it climbs. Being 10% out shows up as a position that drifts from reality in the middle of the travel and snaps back at the end stops, where it recalibrates. *)
    T_TravelDown : TIME := TIME#20s0ms;
    T_Lockout : TIME := TIME#1s0ms;  (* Dead time between a stop and starting the other direction, so a reversing contactor is never asked to change its mind while the motor is still turning. *)
    T_EndStop : TIME := TIME#2s0ms;  (* How long the motor keeps running once it should have reached an end stop. A full OPEN or CLOSE does not trust the estimate at all: it runs for the whole travel time plus this margin, from wherever the cover is thought to be. That is what makes every full command a re-reference rather than a journey computed from a number that may be wrong - an estimate cannot heal itself if the length of the run is derived from it. The cost is a motor that runs longer than strictly necessary. The shutter's own end stops and the motor's thermal cutout are what make that safe, and it is what FB_OUTPUT_COVER_MQTT has always done on every command. *)
    Tolerance : BYTE := 2;  (* How close to the requested position counts as bArrived, in percent. Below about 2 the cover hunts, because a shutter cannot be positioned finer than its own start and stop time. *)
    PublishStep : BYTE := 5;  (* Percent of travel between position publishes while the cover is moving. Every rStep is one MQTT message; 5 gives a slider that visibly moves without putting twenty messages on the broker per journey. The exact position is always published once movement ends, whatever this is set to. *)
  END_VAR
  VAR_OUTPUT
    MU : BOOL;  (* Motor contactors. Never both TRUE, and never switched straight from one to the other - T_Lockout always passes between them. *)
    MD : BOOL;
    Position : BYTE;  (* How far open, 0 closed to 100 open, the way Home Assistant counts a cover. *)
    Moving : BOOL;  (* A motor is running. *)
    PositionKnown : BOOL;  (* An end stop has been reached since power-up, so the position is measured rather than assumed. FALSE means the cover has not yet been anywhere it could be sure of. *)
  END_VAR
  VAR
    {attribute 'noinit'}
    {attribute 'instance-path'}
    sInstancePath : STRING(GVL_MQTT.MQTT_TOPIC_LEN);  (* object's full instance name *)
    rPositionReal : REAL;  (* --- the position estimate --- Kept as a REAL: a 20 ms task tick against a 20 s travel is 0.1% per cycle, which would round to nothing in a BYTE and the cover would never appear to move at all. *)
    rTarget : REAL;  (* Where the cover has been asked to go, in percent. Zero at power-up, which together with bArrived means "stay put" rather than "close" - see below. *)
    bArrived : BOOL := TRUE;  (* The current rTarget has been satisfied, so nothing should move until something asks again. TRUE at power-up, and that is the whole reason a restart does not send every cover in the building somewhere: a rTarget of 0 with bArrived FALSE would have been read as "close", and a rTarget of 100 as "open", and one of those was in fact what the first bench run did. *)
    iDriving : INT;  (* 0 stopped, 1 iDriving up, -1 iDriving down *)
    iDrivingLast : INT;  (* What iDriving was last cycle, so a direction change can be caught *)
    iManualDrive : INT;  (* A held button overrides the rTarget entirely, and releasing it pins the rTarget to wherever the cover got to. *)
    bReferencing : BOOL;  (* A full-travel command is in progress: drive the whole travel time plus T_EndStop and finish against the physical stop, whatever the estimate says. *)
    fbRefRun : Standard.TON;
    tRefTime : TIME;
    byReported : BYTE;  (* What gets published, which is not always what is estimated: an unreferenced cover never reports exactly 0 or 100, because Home Assistant treats those as the limits and disables the button that would have re-referenced it. *)
    tNow : TIME;
    tLast : TIME;
    bValid : BOOL;
    udiDtMs : UDINT;
    udiTravelMs : UDINT;
    rStep : REAL;
    fbLockout : Standard.TON;
    fbEndStop : Standard.TON;
    bAtEnd : BOOL;
    bMqttRequestOpen : BOOL;  (* --- MQTT --- *)
    bMqttRequestClose : BOOL;
    bMqttRequestStop : BOOL;
    bMqttRequestPosition : BOOL;
    byMqttRequestPositionPct : BYTE;
    sState : STRING(10);
    sPublishedState : STRING(10);
    byPublishedPosition : BYTE;
    bPositionPublished : BOOL;
    bStartup : BOOL := TRUE;
    Payload : STRING(20);
    PositionTopic : STRING(GVL_MQTT.MQTT_TOPIC_LEN);
    SetPositionTopic : STRING(GVL_MQTT.MQTT_TOPIC_LEN);
    iDiff : INT;
  END_VAR
  VAR CONSTANT
    ciDriveStop : INT := 0;
    ciDriveUp : INT := 1;
    ciDriveDown : INT := -1;
    cudiMaxTickMs : UDINT := 500;  (* A cycle longer than this is a debugger breakpoint, a download, or a task overrun - not travel. Integrating it would teleport the cover. *)
  END_VAR

            (* --- self-wiring prologue ----------------------------------------------------
   Set FriendlyName at the declaration and this block wires itself from
   GVL_MQTT on its first cyclic call, then announces itself to Home
   Assistant. Same idiom, and the same reasons, as every other block here: see
   FB_OUTPUT_COVER_MQTT.

   It shares the cover prefix and the cover collector with that block. Nothing
   distinguishes the two on the wire - both are covers, and the collector asks
   every registered instance whether a message is theirs.

   A block wired this way MUST be called cyclically. An instance whose body never
   runs stays unwired and never appears in Home Assistant, and nothing warns
   about it. *)
IF FriendlyName <> '' THEN

	IF NOT bInitMqttDone THEN
		THIS^.InitMqtt(
			MQTTPublishPrefix := ADR(GVL_MQTT.MqttPubCoverPrefix),
			MQTTSubscribePrefix := ADR(GVL_MQTT.MqttSubCoverPrefix),
			pMqttPublishQueue := ADR(GVL_MQTT.fbMqttPublishQueue),
			pMqttCallbackCollector := ADR(GVL_MQTT.collector_FB_OUTPUT_COVER_MQTT));
	END_IF

	IF bInitMqttDone AND NOT bInitMqttDiscoveryDone THEN
		THIS^.InitMqttDiscovery(
			Device := ADR(GVL_MQTT.PLC_Device),
			Name := FriendlyName);
	END_IF

END_IF

IF bInitMqttDone AND (PositionTopic = '') THEN
	PositionTopic := CONCAT(THIS^.sMQTTPublishTopic, '/POSITION');
	SetPositionTopic := CONCAT(THIS^.sMQTTSubscribeTopic, '/POSITION');
END_IF

(* --- how much time has passed -------------------------------------------------
   The position is integrated from run time, so the length of a cycle is the one
   measurement this block cannot do without. A tick longer than cudiMaxTickMs is a
   download, a breakpoint or a task overrun rather than travel, and is dropped:
   integrating it would teleport the cover. *)
tNow := TIME();
IF NOT bValid THEN
	bValid := TRUE;
	udiDtMs := 0;
ELSE
	udiDtMs := TIME_TO_UDINT(tNow) - TIME_TO_UDINT(tLast);
	IF udiDtMs > cudiMaxTickMs THEN
		udiDtMs := 0;
	END_IF
END_IF
tLast := tNow;

(* --- integrate ---------------------------------------------------------------
   Whatever the motor did last cycle is what moved the cover, so the estimate is
   advanced before this cycle's decision is taken. *)
IF iDriving = ciDriveUp THEN
	udiTravelMs := TIME_TO_UDINT(T_TravelUp);
	IF udiTravelMs > 0 THEN
		rStep := UDINT_TO_REAL(udiDtMs) * 100.0 / UDINT_TO_REAL(udiTravelMs);
		rPositionReal := rPositionReal + rStep;
	END_IF
ELSIF iDriving = ciDriveDown THEN
	udiTravelMs := TIME_TO_UDINT(T_TravelDown);
	IF udiTravelMs > 0 THEN
		rStep := UDINT_TO_REAL(udiDtMs) * 100.0 / UDINT_TO_REAL(udiTravelMs);
		rPositionReal := rPositionReal - rStep;
	END_IF
END_IF

IF rPositionReal > 100.0 THEN
	rPositionReal := 100.0;
END_IF
IF rPositionReal < 0.0 THEN
	rPositionReal := 0.0;
END_IF

(* --- a held button wins -------------------------------------------------------
   A person watching the cover beats anything Home Assistant asked for, and beats
   it by abandoning the rTarget rather than queueing behind it: releasing the
   button pins the rTarget to wherever the cover got to, so nothing resumes.

   Both buttons at once is not a command. There is no sane guess to make. *)
IF UP AND NOT DN THEN
	iManualDrive := ciDriveUp;
ELSIF DN AND NOT UP THEN
	iManualDrive := ciDriveDown;
ELSE
	IF iManualDrive <> ciDriveStop THEN
		rTarget := rPositionReal;
		bArrived := TRUE;
		bReferencing := FALSE;
	END_IF
	iManualDrive := ciDriveStop;
END_IF

(* --- and what Home Assistant asked for ---------------------------------------
   Latched by the callback, consumed here, so a command that arrives mid-cycle is
   acted on exactly once. *)
IF bMqttRequestStop THEN
	bMqttRequestStop := FALSE;
	(* Hold here. The rTarget has to be dragged to the present position or the
	   interrupted journey would resume on the next cycle - a stop that only
	   pauses is not a stop. *)
	rTarget := rPositionReal;
	bArrived := TRUE;
	bReferencing := FALSE;
ELSIF bMqttRequestOpen THEN
	bMqttRequestOpen := FALSE;
	rTarget := 100.0;
	bArrived := FALSE;
	bReferencing := TRUE;
ELSIF bMqttRequestClose THEN
	bMqttRequestClose := FALSE;
	rTarget := 0.0;
	bArrived := FALSE;
	bReferencing := TRUE;
ELSIF bMqttRequestPosition THEN
	bMqttRequestPosition := FALSE;
	rTarget := BYTE_TO_REAL(byMqttRequestPositionPct);
	bArrived := FALSE;
	(* A slider dragged to either extreme is a full-travel command like any other,
	   and gets the same re-reference. *)
	bReferencing := (rTarget >= 100.0) OR (rTarget <= 0.0);
END_IF

